               3:  //M003_GENERATE_ALERT
                   #methodInputs := REF("MII_Interface_Data".MII_METHODS."M003_GENERATE_ALERT".Inputs);
                   VariantPut(SRC := "MII_Interface_Data".MII_METHODS."M003_GENERATE_ALERT".Inputs,
                              DST := #methodInputs);
                   #methodOutputs := REF("MII_Interface_Data".MII_METHODS."M003_GENERATE_ALERT".Outputs);
                   VariantPut(SRC := "MII_Interface_Data".MII_METHODS."M003_GENERATE_ALERT".Outputs,
                              DST := #methodOutputs);

               4:  //M102_REWORK_DECLARATION
                   #methodInputs := REF("MII_Interface_Data".MII_METHODS."M102_REWORK_DECLARATION".Inputs);
                   VariantPut(SRC := "MII_Interface_Data".MII_METHODS."M102_REWORK_DECLARATION".Inputs,
                              DST := #methodInputs);
                   #methodOutputs := REF("MII_Interface_Data".MII_METHODS."M102_REWORK_DECLARATION".Outputs);
                   VariantPut(SRC := "MII_Interface_Data".MII_METHODS."M102_REWORK_DECLARATION".Outputs,
                              DST := #methodOutputs);

               5:  //M002_GET_PLANTS
                   #methodOutputs := REF("MII_Interface_Data".MII_METHODS."M002_GET_PLANTS".Outputs);
                   VariantPut(SRC := "MII_Interface_Data".MII_METHODS.M002_GET_PLANTS.Outputs,
                              DST := #methodOutputs);

               6: //NON TRS
                   #methodInputs := REF("MII_Interface_Data".MII_METHODS.M004_NTRS.Inputs);
                   VariantPut(SRC := "MII_Interface_Data".MII_METHODS.M004_NTRS.Inputs,
                              DST := #methodInputs);
                   #methodOutputs := REF("MII_Interface_Data".MII_METHODS.M004_NTRS.Outputs);
                   VariantPut(SRC := "MII_Interface_Data".MII_METHODS.M004_NTRS.Outputs,
                              DST := #methodOutputs);

               7: //PY
                   #methodInputs := REF("MII_Interface_Data".MII_METHODS.M103_PY.Inputs);
                   VariantPut(SRC := "MII_Interface_Data".MII_METHODS.M103_PY.Inputs,
                              DST := #methodInputs);
                   #methodOutputs := REF("MII_Interface_Data".MII_METHODS.M103_PY.Outputs);
                   VariantPut(SRC := "MII_Interface_Data".MII_METHODS.M103_PY.Outputs,
                              DST := #methodOutputs);

               8: //VARABILITY
                   #methodInputs := REF("MII_Interface_Data".MII_METHODS.M005_VARIABILITY.Inputs);
                   VariantPut(SRC := "MII_Interface_Data".MII_METHODS.M005_VARIABILITY.Inputs,
                              DST := #methodInputs);
                   #methodOutputs := REF("MII_Interface_Data".MII_METHODS.M005_VARIABILITY.Outputs);
                   VariantPut(SRC := "MII_Interface_Data".MII_METHODS.M005_VARIABILITY.Outputs,
                              DST := #methodOutputs);


           END_CASE;
       END_REGION ;
   END_IF;
END_REGION

REGION Network 3: Call client fb
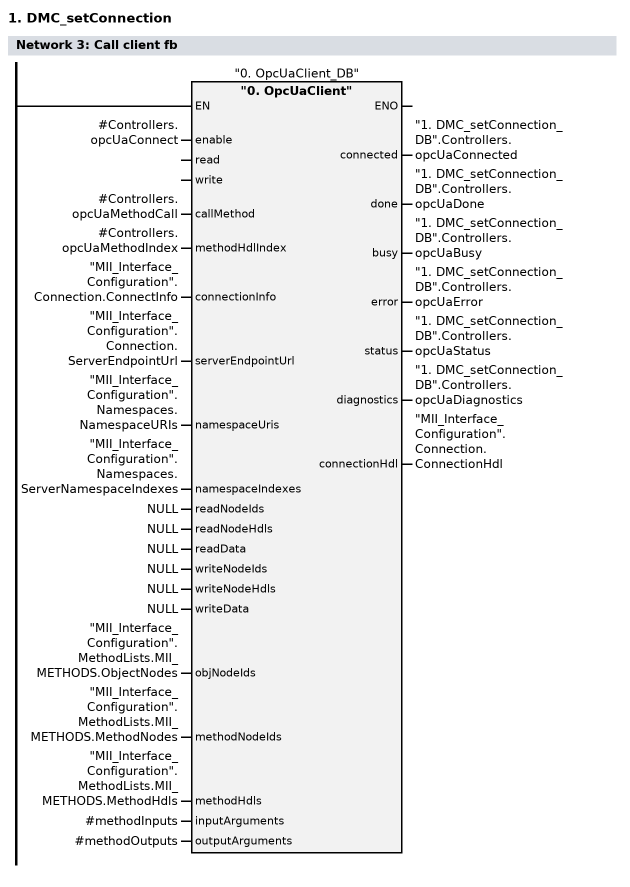
   RUNG wire#powerrail
      "0. OpcUaClient_DB"(enable := #Controllers.opcUaConnect, read :=, write :=, callMethod := #Controllers.opcUaMethodCall, methodHdlIndex := #Controllers.opcUaMethodIndex, connectionInfo := "MII_Interface_Configuration".Connection.ConnectInfo, serverEndpointUrl := "MII_Interface_Configuration".Connection.ServerEndpointUrl, namespaceUris := "MII_Interface_Configuration".Namespaces.NamespaceURIs, namespaceIndexes := "MII_Interface_Configuration".Namespaces.ServerNamespaceIndexes, readNodeIds := NULL, readNodeHdls := NULL, readData := NULL, writeNodeIds := NULL, writeNodeHdls := NULL, writeData := NULL, objNodeIds := "MII_Interface_Configuration".MethodLists.MII_METHODS.ObjectNodes, methodNodeIds := "MII_Interface_Configuration".MethodLists.MII_METHODS.MethodNodes, methodHdls := "MII_Interface_Configuration".MethodLists.MII_METHODS.MethodHdls, inputArguments := #methodInputs, outputArguments := #methodOutputs, connected => "1. DMC_setConnection_DB".Controllers.opcUaConnected, done => "1. DMC_setConnection_DB".Controllers.opcUaDone, busy => "1. DMC_setConnection_DB".Controllers.opcUaBusy, error => "1. DMC_setConnection_DB".Controllers.opcUaError, status => "1. DMC_setConnection_DB".Controllers.opcUaStatus, diagnostics => "1. DMC_setConnection_DB".Controllers.opcUaDiagnostics, connectionHdl => "MII_Interface_Configuration".Connection.ConnectionHdl)
   END_RUNG
   // the same network as SCL:
   "0. OpcUaClient_DB"(enable := #Controllers.opcUaConnect,   // "0. OpcUaClient"
                       callMethod := #Controllers.opcUaMethodCall,
                       methodHdlIndex := #Controllers.opcUaMethodIndex,
                       connectionInfo := "MII_Interface_Configuration".Connection.ConnectInfo,
                       serverEndpointUrl := "MII_Interface_Configuration".Connection.ServerEndpointUrl,
                       namespaceUris := "MII_Interface_Configuration".Namespaces.NamespaceURIs,
                       namespaceIndexes := "MII_Interface_Configuration".Namespaces.ServerNamespaceIndexes,
                       readNodeIds := NULL,
                       readNodeHdls := NULL,
                       readData := NULL,
                       writeNodeIds := NULL,
                       writeNodeHdls := NULL,
                       writeData := NULL,
                       objNodeIds := "MII_Interface_Configuration".MethodLists.MII_METHODS.ObjectNodes,
                       methodNodeIds := "MII_Interface_Configuration".MethodLists.MII_METHODS.MethodNodes,
                       methodHdls := "MII_Interface_Configuration".MethodLists.MII_METHODS.MethodHdls,
                       inputArguments := #methodInputs,
                       outputArguments := #methodOutputs,
                       connected => "1. DMC_setConnection_DB".Controllers.opcUaConnected,
                       done => "1. DMC_setConnection_DB".Controllers.opcUaDone,
                       busy => "1. DMC_setConnection_DB".Controllers.opcUaBusy,
                       error => "1. DMC_setConnection_DB".Controllers.opcUaError,
                       status => "1. DMC_setConnection_DB".Controllers.opcUaStatus,
                       diagnostics => "1. DMC_setConnection_DB".Controllers.opcUaDiagnostics,
                       connectionHdl => "MII_Interface_Configuration".Connection.ConnectionHdl);
END_REGION

REGION Network 4 (SCL): Post method call
   IF #Controllers.opcUaMethodCall AND (#Controllers.opcUaDone OR #Auxiliar.timeout) THEN
       REGION SWITCH CASE
           CASE #Controllers.opcUaMethodIndex OF
               0:  //M000_PRODUCTION_DECLARATION
                   //Send the inputs and the output to the HMI
                   "MII_Parameters".M000_Status.Inputs := "MII_Interface_Data".MII_METHODS.M000_PRODUCTION_DECLARATION.Inputs;
                   "MII_Parameters".M000_Status.Outputs := "MII_Interface_Data".MII_METHODS.M000_PRODUCTION_DECLARATION.Outputs;


                   IF "MII_Interface_Data".MII_METHODS.M000_PRODUCTION_DECLARATION.Outputs.SUCCESS_FLAG = 0 OR #Auxiliar.timeout THEN
                       //Write error status
                       IF #Auxiliar.timeout THEN
                           "MII_Parameters".M000_Status.status := Wstring#'TimeoutERROR';
                       ELSE
                           "MII_Parameters".M000_Status.status := "MII_Interface_Data".MII_METHODS.M000_PRODUCTION_DECLARATION.Outputs.STATUS_MESSAGE;
                       END_IF;

                       //Get error timestamp 
                       #retVal := RD_LOC_T("MII_Parameters".M000_Status.timestamp);

                       //Set error trigger to HMI store values
                       //Note: HMI must reset this tag after writing the file
                       "MII_Parameters".M000_Status.error := TRUE;
                   ELSE
                       //Reset error if declaration is ok
                       "MII_Parameters".M000_Status.error := FALSE;
                       "MII_Parameters".M000_Status.status := "MII_Interface_Data".MII_METHODS.M000_PRODUCTION_DECLARATION.Outputs.STATUS_MESSAGE;
                   END_IF;

                   //Reset test command and add one to the auxiliar cycle counter
                   IF "MII_Parameters".Commands.testProdDeclaration THEN
                       "MII_Parameters".Commands.testProdDeclaration := FALSE;
                       "MII_Parameters".Commands.auxTestProdDeclaration := "MII_Parameters".Commands.auxTestProdDeclaration + 1;
                   END_IF;

               1: //M002_GET_LOCAL_TIME
                   IF #Auxiliar.timeout THEN
                       "MII_Parameters".M002_Status.status := WSTRING#'TimeoutERROR';
                   ELSE
                       //Overwrite system time
                       #retVal := WR_LOC_T(LOCTIME := "MII_Interface_Data".MII_METHODS.M001_GET_LOCAL_TIME.Outputs.DATETIME_LOCAL, DST := TRUE);

                       //Set M002_status
                       "MII_Parameters".M002_Status.localTime := "MII_Interface_Data".MII_METHODS.M001_GET_LOCAL_TIME.Outputs.DATETIME_LOCAL;
                       "MII_Parameters".M002_Status.status := WSTRING#'OK';

                       //Reset command after calling the method
                       "MII_Parameters".Commands.getLocalTime := FALSE;
                   END_IF;

               2: //TO BE DEVELOPED
                   ;

               3: //TO BE DEVELOPED
                   ;

               4: //TO BE DEVELOPED
                   ;

               5: //TO BE DEVELOPED
                   ;

               6: //TO BE DEVELOPED
                   ;

               7: //TO BE DEVELOPED
                   ;

               8: //TO BE DEVELOPED
                   ;

           END_CASE;
       END_REGION

       //RESET METHOD INDEX
       #CallBuffer[#Controllers.opcUaMethodIndex] := FALSE;

       //RESET METHOD TAG
       #Controllers.opcUaMethodCall := FALSE;
   END_IF;
END_REGION

REGION Network 5 (SCL): Device diagnostics
   // Read diagnostic status
   "MII_Parameters".Connection_Status.opcUaConnected := #Controllers.opcUaConnected;
   "MII_Parameters".Connection_Status.opcUaError := #Controllers.opcUaError;
   "MII_Parameters".Connection_Status.opcUaStatus := #Controllers.opcUaStatus;
   "MII_Parameters".Connection_Status.opcUaDiagnostics := #Controllers.opcUaDiagnostics.subfunctionStatus;

   // Shift data to display on HMI
   IF #Controllers.opcUaDiagnostics.subfunctionStatus > 65536 THEN
       "MII_Parameters".Connection_Status.aux.opcUaSubfunctionStatus := SHR(IN := #Controllers.opcUaDiagnostics.subfunctionStatus, N := 16);
   END_IF;

   // Output error parameters
   IF NOT #Controllers.opcUaError THEN
       CASE #Controllers.opcUaStatus OF
           16#0000:
               IF NOT #Controllers.opcUaDone THEN
                   //Client not connected.
                   "MII_Parameters".Connection_Status.aux.diagnosticStatus := 1;
               ELSE
                   //Job successfully executed.
                   "MII_Parameters".Connection_Status.aux.diagnosticStatus := 2;
               END_IF;

           16#7000:
               IF NOT #Controllers.opcUaDone THEN
                   //Client connected and ready for job.
                   "MII_Parameters".Connection_Status.aux.diagnosticStatus := 3;
               ELSE
                   //Connection successfully established and ready for job.
                   "MII_Parameters".Connection_Status.aux.diagnosticStatus := 4;
               END_IF;

           16#7001: //Job is running.
               "MII_Parameters".Connection_Status.aux.diagnosticStatus := 5;
       END_CASE;
   ELSE
       // Output parameters with error
       "MII_Parameters".Connection_Status.aux.diagnosticStatus := #Controllers.opcUaStatus;

       // Automatically manage the 16#80AE_0000 error
       IF NOT "MII_Parameters".Commands.forceReconnection AND NOT "MII_Parameters".Connection_Status.opcUaConnected THEN
           // Forces the reconnection
           "MII_Parameters".Commands.forceReconnection := TRUE;

           IF "0. OpcUaClient_DB".statOpcUaRequests.disconnect THEN
               // Reset disconnect button 
               "0. OpcUaClient_DB".statOpcUaRequests.disconnect := FALSE;
           END_IF;
       END_IF;
   END_IF;
END_REGION

REGION Network 6 (SCL): Try to call method again routine
   // //Method call timeout
   // #Timers.tryAgain(IN := "MII_Parameters".M000_Status.error,
   //                  PT := t#2s,
   //                  Q => #Auxiliar.tryAgain);

   // IF #Controllers.opcUaConnected AND #Auxiliar.tryAgain THEN
   //              //Try again
   //              IF NOT #CallBuffer[0] THEN
   //                  #CallBuffer[0] := TRUE;

   //                  //Add one attempt to counter
   //                  "MII_Parameters".Connection_Status.aux.nAttemptsTotal := "MII_Parameters".Connection_Status.aux.nAttemptsTotal + 1;
   //              END_IF;

   //              //Restart timer
   //              RESET_TIMER(#Timers.tryAgain);

   //          END_IF;
END_REGION
END_FUNCTION_BLOCK

FUNCTION_BLOCK "0. OpcUaClient"
TITLE = OpcUaClient
{ S7_Optimized_Access := 'FALSE' }
AUTHOR : SiemensAG
VERSION : 1.3
//OPC UA-Client-Wrapper
   VAR_INPUT 
      enable : Bool;   // TRUE: Enable connection to OPC UA server
      read : Bool;   // TRUE: Execute Read functionality
      write : Bool;   // TRUE: Execute Write functionality
      callMethod : Bool;   // TRUE: Execute Method Call
      methodHdlIndex : SInt;   // Index of method in "methodHdls" that should be called
      connectionInfo {InstructionName := 'OPC_UA_SessionConnectInfo'; LibVersion := '1.0'} : OPC_UA_SessionConnectInfo;   // Connection Information for session establishment to OPC UA server
      serverEndpointUrl : String;   // Endpoint of OPC UA server
   END_VAR

   VAR_OUTPUT 
      connected { ExternalWritable := 'False'} : Bool;   // TRUE: Connection to OPC UA server is established and valid
      done { ExternalWritable := 'False'} : Bool;   // TRUE: Functions Read, Write or Method Call were executed successfully
      busy { ExternalWritable := 'False'} : Bool;   // TRUE: FB is working
      error { ExternalWritable := 'False'} : Bool;   // TRUE: FB is in faulty state
      status { ExternalWritable := 'False'} : Word;   // 16#0000 - 16#7FFF: Status of the FB, 16#8000 - 16#FFFF: Error identification
      diagnostics { ExternalWritable := 'False'} : "typeFbDiagnostics";   // Diagnostics information of FB when error occurs
      connectionHdl { ExternalWritable := 'False'} : DWord;   // Connection handle which is used for OPC UA connection to the server
   END_VAR

   VAR_IN_OUT 
      namespaceUris : Variant;   // Pointer to the Namespace URIs of the OPC UA client interface (NULL if not used)
      namespaceIndexes : Variant;   // Pointer to the Namespace Indexes of the OPC UA client interface (NULL if not used)
      readNodeIds : Variant;   // Pointer to the Node-IDs of the nodes to read of the OPC UA client interface (NULL if not used)
      readNodeHdls : Variant;   // Pointer to the Node handles of the registered nodes to read of the OPC UA client interface (NULL if not used)
      readData : Variant;   // Pointer to the storage area for read data (NULL if not used)
      writeNodeIds : Variant;   // Pointer to the Node-IDs of the nodes to write of the OPC UA client interface (NULL if not used)
      writeNodeHdls : Variant;   // Pointer to the Node handles of the registered nodes to write of the OPC UA client interface (NULL if not used)
      writeData : Variant;   // Pointer to the storage area for write data (NULL if not used)
      objNodeIds : Variant;   // Pointer to the Node-IDs of the method objects (instance DB) of the OPC UA client interface (NULL if not used)
      methodNodeIds : Variant;   // Pointer to the Node-IDs of the methods of the OPC UA client Interface (NULL if not used)
      methodHdls : Variant;   // Pointer to the Node handles of the registered methods of the OPC UA client interface (NULL if not used)
      inputArguments : Variant;   // Pointer to the Input Arguments of the called method (NULL if not used)
      outputArguments : Variant;   // Pointer to the Output Arguments of the called method (NULL if not used)
   END_VAR

   VAR 
      instOpcUaConnect {InstructionName := 'OPC_UA_Connect'; LibVersion := '1.0'; ExternalAccessible := 'False'; ExternalVisible := 'False'; ExternalWritable := 'False'} : OPC_UA_Connect;
      instOpcUaConnectionGetStatus {InstructionName := 'OPC_UA_ConnectionGetStatus'; LibVersion := '1.0'; ExternalAccessible := 'False'; ExternalVisible := 'False'; ExternalWritable := 'False'} : OPC_UA_ConnectionGetStatus;
      instOpcUaNamespaceGIL {InstructionName := 'OPC_UA_NamespaceGetIndexList'; LibVersion := '1.0'; ExternalAccessible := 'False'; ExternalVisible := 'False'; ExternalWritable := 'False'} : OPC_UA_NamespaceGetIndexList;
      InstOpcUaGHLRead {InstructionName := 'OPC_UA_NodeGetHandleList'; LibVersion := '1.0'; ExternalAccessible := 'False'; ExternalVisible := 'False'; ExternalWritable := 'False'} : OPC_UA_NodeGetHandleList;
      instOpcUaGHLWrite {InstructionName := 'OPC_UA_NodeGetHandleList'; LibVersion := '1.0'; ExternalAccessible := 'False'; ExternalVisible := 'False'; ExternalWritable := 'False'} : OPC_UA_NodeGetHandleList;
      instOpcUaGHLMethods {InstructionName := 'OPC_UA_MethodGetHandleList'; LibVersion := '1.0'; ExternalAccessible := 'False'; ExternalVisible := 'False'; ExternalWritable := 'False'} : OPC_UA_MethodGetHandleList;   // Get node handles for Methods
      InstOpcUaRHLRead {InstructionName := 'OPC_UA_NodeReleaseHandleList'; LibVersion := '1.0'; ExternalAccessible := 'False'; ExternalVisible := 'False'; ExternalWritable := 'False'} : OPC_UA_NodeReleaseHandleList;
      instOpcUaRHLWrite {InstructionName := 'OPC_UA_NodeReleaseHandleList'; LibVersion := '1.0'; ExternalAccessible := 'False'; ExternalVisible := 'False'; ExternalWritable := 'False'} : OPC_UA_NodeReleaseHandleList;
      instOpcUaRHLMethods {InstructionName := 'OPC_UA_MethodReleaseHandleList'; LibVersion := '1.0'; ExternalAccessible := 'False'; ExternalVisible := 'False'; ExternalWritable := 'False'} : OPC_UA_MethodReleaseHandleList;
      instOpcUaReadList {InstructionName := 'OPC_UA_ReadList'; LibVersion := '1.0'; ExternalAccessible := 'False'; ExternalVisible := 'False'; ExternalWritable := 'False'} : OPC_UA_ReadList;
      instOpcUaWriteList {InstructionName := 'OPC_UA_WriteList'; LibVersion := '1.0'; ExternalAccessible := 'False'; ExternalVisible := 'False'; ExternalWritable := 'False'} : OPC_UA_WriteList;   // Write values of multiple nodes
      instOpcUaMethodCall {InstructionName := 'OPC_UA_MethodCall'; LibVersion := '1.0'; ExternalAccessible := 'False'; ExternalVisible := 'False'; ExternalWritable := 'False'} : OPC_UA_MethodCall;
      instOpcUaDisconnect {InstructionName := 'OPC_UA_Disconnect'; LibVersion := '1.0'; ExternalAccessible := 'False'; ExternalVisible := 'False'; ExternalWritable := 'False'} : OPC_UA_Disconnect;
      statOldTriggers { ExternalAccessible := 'False'; ExternalVisible := 'False'; ExternalWritable := 'False'} : Struct   // Internal structure for Trigger handling
         connect { ExternalAccessible := 'False'; ExternalVisible := 'False'; ExternalWritable := 'False'} : Bool;   // Saved Trigger for Connection establishment
         reconnect { ExternalAccessible := 'False'; ExternalVisible := 'False'; ExternalWritable := 'False'} : Bool;   // Saved Trigger for Connection reestablishment
         disconnect { ExternalAccessible := 'False'; ExternalVisible := 'False'; ExternalWritable := 'False'; S7_SetPoint := 'True'} : Bool;   // Saved Trigger for disconnecting
         read { ExternalAccessible := 'False'; ExternalVisible := 'False'; ExternalWritable := 'False'; S7_SetPoint := 'True'} : Bool;   // Saved Trigger for Read
         write { ExternalAccessible := 'False'; ExternalVisible := 'False'; ExternalWritable := 'False'; S7_SetPoint := 'True'} : Bool;   // Saved Trigger for Write
         callMethod { ExternalAccessible := 'False'; ExternalVisible := 'False'; ExternalWritable := 'False'} : Bool;   // Saved Trigger for Method Call
         clearSession { ExternalAccessible := 'False'; ExternalVisible := 'False'; ExternalWritable := 'False'} : Bool;   // Saved Trigger for Session Clearing
      END_STRUCT;
      statState { ExternalWritable := 'False'} : Int;   // Actual state of the state machine. 0: connect; 1: get Namespaces; 3: Get List Handles; 4: Connected; 5: Disconnect
      statDone { ExternalAccessible := 'False'; ExternalVisible := 'False'; ExternalWritable := 'False'} : Bool;   // Read, Write, MethodCall finished without error.
      statConnected { ExternalAccessible := 'False'; ExternalVisible := 'False'; ExternalWritable := 'False'} : Bool;   // Connection to OPC UA Server is established and valid.
      statBusy { ExternalVisible := 'False'; ExternalWritable := 'False'} : Bool;   // FB is busy.
      statDiagnostics { ExternalAccessible := 'False'; ExternalVisible := 'False'; ExternalWritable := 'False'} : "typeFbDiagnostics";   // Diagnostic structure for internal use.
      statDiagnosticsEmpty { ExternalWritable := 'False'} : "typeFbDiagnostics";   // Empty diagnostic structure, to initialize Output.
      statOpcUaRequests { ExternalAccessible := 'False'; ExternalVisible := 'False'; ExternalWritable := 'False'} : Struct   // Internal structure for OPC UA function blocks requests.
         connect { ExternalAccessible := 'False'; ExternalVisible := 'False'; ExternalWritable := 'False'} : Bool;   // Request for OPC_UA_Connect
         conGS { ExternalAccessible := 'False'; ExternalVisible := 'False'; ExternalWritable := 'False'} : Bool;   // Request for OPC_UA_ConnectionGetStatus
         NGIL { ExternalAccessible := 'False'; ExternalVisible := 'False'; ExternalWritable := 'False'} : Bool;   // Request for OPC_UA_NamespaceGetIndexList
         readGHL { ExternalAccessible := 'False'; ExternalVisible := 'False'; ExternalWritable := 'False'} : Bool;   // Request for OPC_UA_NodeGetHandleList for ReadList
         methodsGHL { ExternalAccessible := 'False'; ExternalVisible := 'False'; ExternalWritable := 'False'} : Bool;   // Request for OPC_UA_MethodGetHandleList
         writeGHL { ExternalAccessible := 'False'; ExternalVisible := 'False'; ExternalWritable := 'False'} : Bool;   // Request for OPC_UA_NodeGetHandleList for WriteList
         read { ExternalAccessible := 'False'; ExternalVisible := 'False'; ExternalWritable := 'False'} : Bool;   // Request for OPC_UA_ReadList
         write { ExternalAccessible := 'False'; ExternalVisible := 'False'; ExternalWritable := 'False'} : Bool;   // Request for OPC_UA_WriteList
         methodCall { ExternalAccessible := 'False'; ExternalVisible := 'False'; ExternalWritable := 'False'} : Bool;   // Request for OPC_UA_MethodCall
         readRHL { ExternalAccessible := 'False'; ExternalVisible := 'False'; ExternalWritable := 'False'} : Bool;   // Request for OPC_UA_NodeReleaseHandleList for ReadList
         writeRHL { ExternalAccessible := 'False'; ExternalVisible := 'False'; ExternalWritable := 'False'} : Bool;   // Request for OPC_UA_NodeReleaseHandleList for WriteList
         methodsRHL { ExternalAccessible := 'False'; ExternalVisible := 'False'; ExternalWritable := 'False'} : Bool;   // Request for OPC_UA_MethodReleaseHandleList
         disconnect { ExternalAccessible := 'False'; ExternalVisible := 'False'; ExternalWritable := 'False'} : Bool;   // Request for OPC_UA_Disconnect
      END_STRUCT;
      statRegisteredLists { ExternalWritable := 'False'} : Struct   // Internal structure for registered Lists/Namespaces. For Diagnostic purpose.
         NamespaceIndexes { ExternalWritable := 'False'} : Bool;   // Namespace Indexes are registered by OPC_UA_NamespaceGetIndexList
         Read { ExternalWritable := 'False'} : Bool;   // Read list is registered by OPC_UA_NodeGetHandleList
         Write { ExternalWritable := 'False'} : Bool;   // Write list is registered by OPC_UA_NodeGetHandleList
         Methods { ExternalWritable := 'False'} : Bool;   // Method list is registered by OPC_UA_MethodGetHandleList
      END_STRUCT;
      statDiagCounter { ExternalWritable := 'False'} : Struct   // Internal structure for counting connects/registrations/functions. For Diagnostic purpose.
         Connect { ExternalVisible := 'False'; ExternalWritable := 'False'} : UInt;   // Counter for successful connects or reconnects.
         NamespaceReg { ExternalWritable := 'False'} : UInt;   // Counter for successful Namespace registrations.
         RegisterRead { ExternalWritable := 'False'} : UInt;   // Counter for successful Read List registrations.
         RegisterWrite { ExternalWritable := 'False'} : UInt;   // Counter for successful Write List registrations.
         RegisterMethods { ExternalWritable := 'False'} : UInt;   // Counter for successful Method List registrations.
         Read { ExternalWritable := 'False'} : UInt;   // Counter for successful Read function executions.
         Write { ExternalWritable := 'False'} : UInt;   // Counter for successful Write function executions.
         MethodCall { ExternalWritable := 'False'} : UInt;   // Counter for successful Method Calls.
      END_STRUCT;
      statMethodResult { ExternalWritable := 'False'} : DWord;   // OPC UA result after Method Call.
      statMethodHdl { ExternalAccessible := 'False'; ExternalVisible := 'False'; ExternalWritable := 'False'} : DWord;   // Calculated Method Handle. Dependend on INPUT: methodHdlIndex.
      statMethodHdlId { ExternalAccessible := 'False'; ExternalVisible := 'False'; ExternalWritable := 'False'} : DInt;   // Internal Variable for INPUT: methodHdlIndex.
      statConnectionHdl { ExternalAccessible := 'False'; ExternalVisible := 'False'; ExternalWritable := 'False'} : DWord;   // Internal Variable for Connection Handle.
      statRHLTrigger { ExternalAccessible := 'False'; ExternalVisible := 'False'; ExternalWritable := 'False'} : Bool;   // Trigger, do start with releasing Lists for disconnect.
      statCheckConnectionStatus { ExternalAccessible := 'False'; ExternalVisible := 'False'; ExternalWritable := 'False'} : Bool;   // If TRUE, OPC_UA_ConnectionGetStatus is called to diagnose the connection.
      statCycDiagTrigger { ExternalAccessible := 'False'; ExternalVisible := 'False'; ExternalWritable := 'False'} : Bool;   // Cyclic trigger for OPC_UA_ConnectionGetStatus-
      instCycDiag {InstructionName := 'IEC_TIMER'; LibVersion := '1.0'; ExternalAccessible := 'False'; ExternalVisible := 'False'; ExternalWritable := 'False'} : IEC_TIMER;   // Timer for cyclic connection diagnostics.
      statOpcUaReadTimeStamps { ExternalWritable := 'False'} : Array[0..299] of LDT;   // Timestamps of read variables. For diagnostic purpose.
      statSerializeMethodHdls { ExternalAccessible := 'False'; ExternalVisible := 'False'; ExternalWritable := 'False'} : Array[0..1199] of Byte;   // Array for calculating the MethodHdl together with the INPUT methodHdlIndex.
      statOpcUaStatusLists { ExternalWritable := 'False'} : Struct   // Internal structure for Status Lists, that are used by every OPC_UA_xxx FB
         methodRHL { ExternalWritable := 'False'} : Array[0..299] of DWord;   // Status List for Method OPC_UA_ReleaseHandleList
         methodGHL { ExternalWritable := 'False'} : Array[0..299] of DWord;   // Status List for Method OPC_UA_GetHandleList
         writeRHL { ExternalWritable := 'False'} : Array[0..299] of DWord;   // Status List for Write OPC_UA_ReleaseHandleList
         writeList { ExternalWritable := 'False'} : Array[0..299] of DWord;   // Status List for Write OPC_UA_WritedList
         writeGHL { ExternalWritable := 'False'} : Array[0..299] of DWord;   // Status List for WriteOPC_UA_GetHandleList
         readRHL { ExternalWritable := 'False'} : Array[0..299] of DWord;   // Status List for Read OPC_UA_ReleaseHandleList
         readList { ExternalWritable := 'False'} : Array[0..299] of DWord;   // Status List for Read OPC_UA_ReadList
         readGHL { ExternalWritable := 'False'} : Array[0..299] of DWord;   // Status List for Read OPC_UA_GetHandleList
         namespaceGIL { ExternalWritable := 'False'} : Array[0..299] of DWord;   // Status List for Namespace OPC_UA_NamespaceGetIndexList
      END_STRUCT;
   END_VAR

   VAR_TEMP 
      tempIndex : Int;   // Index for finding errors in statOpcUaStatusLists.
      tempRetVal : Int;   // Return value for Serialize function, that is used for calculating statMethodHdl.
      tempConnectTrigger : Bool;   // Temporary trigger for connection establishment.
      tempDisconnectTrigger : Bool;   // Temporary trigger for disconnect.
      tempReadTrigger : Bool;   // Temporary trigger for Read function.
      tempWriteTrigger : Bool;   // Temporary trigger for Write function.
      tempMethodCallTrigger : Bool;   // Temporary trigger for Method Calls.
      tempReconnectTrigger : Bool;   // Temporary trigger for reconnect.
      tempClearSessionTrigger : Bool;   // Temporary trigger for clean up Session.
   END_VAR

   VAR CONSTANT 
      STATE_CONNECT : Int := 0;   // State for idling until INPUT enable is triggered, to establish a connection.
      STATE_NAMESPACE_GET_INDEX_LIST : Int := 1;   // State for getting Namespace indexes.
      STATE_NODE_GET_HANDLE_LIST : Int := 3;   // State for registration of Read/Write/Method Lists
      STATE_CONNECTED : Int := 4;   // State for idling until INPUT read/write/methodCall has positive edge, to execute function.
      STATE_DISCONNECT : Int := 5;   // State for releasing Read/Write/Method Lists and disconnect.
      CGS_CONNECTED : UDInt := 0;   // OPC_UA_ConnectionGetStatus Connection state is connected.
      CGS_CONN_ERROR : UDInt := 1;   // OPC_UA_ConnectionGetStatus Connection state is in error.
      CGS_SHUTDOWN : UDInt := 2;   // OPC_UA_ConnectionGetStatus Connection state is in shutdown, nodes have to be released and connection terminated.
      CGS_SS_RUNNING : UDInt := 0;   // OPC_UA_ConnectionGetStatus Server state is running.
      CGS_SL_GOOD : Byte := 16#FF;   // OPC_UA_ConnectionGetStatus Connection state is connected.
      STATUS_SESSION_CLEANEDUP : DWord := 16#A000_0105;   // OPC_UA_ConnectionGetStatus: Session is cleaned up and has to be reconnected.
      STATUS_SERVER_NOT_CONNECTED : DWord := 16#800D_0000;   // OPC_UA_ConnectionGetStatus: Choosen Server is not connected.
      STATUS_BAD_CONNECTION_CLOSED : DWord := 16#80AE_0000;   // OPC_UA_ConnectionGetStatus
      STATUS_BUSY : Word := 16#7001;   // Function block is busy.
      STATUS_IDLE : Word := 16#7000;   // Function block idles.
      STATUS_NOT_REGISTERED : Word := 16#80FF;   // Read/Write/Method List is not registered
      STATUS_DONE : Word := 16#0000;   // Read/Write/Method Call was successfully executed.
      CYC_TIME_GCS : Time := T#5S;   // Time for cylic call of OPC_UA_ConnectionGetStatus
      OPC_UA_FUNCTIONS_TIMEOUT : Time := T#10S;   // Timout for all OPC UA Client Function blocks
      ERR_CONNECT : Word := 16#8601;   // Error during connect.
      ERR_NGIL : Word := 16#8602;   // Error during getting Namespace Indexes
      ERR_NGIL_SL : Word := 16#8617;   // Error in Namespace indexes Status list
      ERR_R_GHL : Word := 16#8631;   // Error during Read list registration
      ERR_R_GHL_SL : Word := 16#8731;   // Error in Read handle list Status list
      ERR_W_GHL : Word := 16#8632;   // Error during Write list registration
      ERR_W_GHL_SL : Word := 16#8732;   // Error in Write handle list Status list
      ERR_M_GHL : Word := 16#8633;   // Error during Method list registration
      ERR_M_GHL_SL : Word := 16#8733;   // Error in Method handle List status list
      ERR_RL : Word := 16#8604;   // Error during Read List execution
      ERR_RL_NOTREG : Word := 16#86F4;   // Error, because no Read List is registered, but Read execution was triggered
      ERR_RL_SL : Word := 16#8614;   // Error in Read list status list.
      ERR_WL : Word := 16#8605;   // Error during Write List execution
      ERR_WL_NOTREG : Word := 16#86F5;   // Error, because no Write List is registered, but Write execution was triggered
      ERR_WL_SL : Word := 16#8615;   // Error in Write list status list
      ERR_MC : Word := 16#8606;   // Error durging Method Call execution
      ERR_MC_NOTREG : Word := 16#86F6;   // Error, because no Method List is registered, but Method call execution was triggered
      ERR_MC_SERIALIZE : Word := 16#8616;   // Error during MethodHdl calculation, in Serialize function
      ERR_MC_RESULT : Word := 16#8626;   // Error, that was reported by Methods OPC UA result
      ERR_R_RHL : Word := 16#8671;   // Error during release of Read List
      ERR_R_RHL_SL : Word := 16#8771;   // Error in Release Read List status list
      ERR_W_RHL : Word := 16#8672;   // Error during realease of Write list
      ERR_W_RHL_SL : Word := 16#8772;   // Error in Release Write List status list
      ERR_M_RHL : Word := 16#8673;   // Error during relaese of Method List
      ERR_M_RHL_SL : Word := 16#8773;   // Error in Release Method List status List
      ERR_DISCON : Word := 16#8608;   // Error during disconnect.
      ERR_CGS : Word := 16#8610;   // Error in OPC_UA_ConnectionGetStatus
      ERR_CGS_CSTATE : Word := 16#8611;   // Error in OPC_UA_ConnectionGetStatus, regarding Connection Status
      ERR_CGS_CSTATE_SHUTDOWN : Word := 16#8711;   // Error in OPC_UA_ConnectionGetStats, Connection was shut down
      ERR_CGS_SSTATE : Word := 16#8612;   // Error in OPC_UA_ConnectionGetStatus, regarding Server State
      ERR_CGS_SLVL : Word := 16#8613;   // Error in OPC_UA_ConnectionGetStatus, regarding Service Level
      MAX_LIST_LENGTH : UInt := 299;   // Maximum lenth of Write/Readlist
      MAX_LENGTH_METHOD_INDEX : UInt := 399;   // maximum length of MethodHdls (mas 100 Methods per MethodList)
   END_VAR


BEGIN
	//=============================================================================
	// Siemens AG (c)Copyright (2019)
	//-----------------------------------------------------------------------------
	// Library: -
	// Tested with: CPU 1516-3 PN/DP;  FW 2.8
	// Engineering: TIA Portal (V16)
	// Restrictions: -
	// Requirements: OPC UA Client activated, Fimware V2.8; Set PLC time
	// Functionality: Encapsulates OPC UA client blocks for read, write and method
	//                call including connection handling and diagnosis
	//-----------------------------------------------------------------------------
	// Change log table:
	// Version    Date         Expert in charge           Changes applied
	// 01.00.00   01.02.2019   Siemens SUP Applications   First released version
	// 01.01.00   31.11.2019   Siemens SUP Applications   Interface, Styleguide and user program performance changes
	// 01.02.00   15.10.2020   Siemens SUP Applications   Bugfixes
	// 01.03.00   28.07.2021   Siemens SUP Applications   Fixed RHL issues
	//=============================================================================
	
	
	//State machine
	CASE #statState OF
	  #STATE_CONNECT:
	    REGION Connection Handling
	      //initialize FB
	      IF NOT #enable THEN
	        #statBusy := FALSE;
	        #statDone := FALSE;
	        #statDiagnostics := #statDiagnosticsEmpty;
	        #statOldTriggers.connect := FALSE;
	        #statConnected := FALSE;
	        #statDiagnostics.status := #STATUS_DONE;
	      END_IF;
	      
	      //Rising Edge detection of connect
	      #tempConnectTrigger := #enable AND NOT #statOldTriggers.connect;
	      #statOldTriggers.connect := #enable;
	      //Rising Edge detection for Reconnect functionality
	      #tempReconnectTrigger := #enable AND NOT #statConnected
	      // AND (#statDiagnostics.subfunctionStatus = #STATUS_SESSION_CLEANEDUP
	      // OR #statDiagnostics.subfunctionStatus = #STATUS_BAD_CONNECTION_CLOSED)
	      AND #statDiagnostics.subfunctionStatus = UDINT_TO_DWORD(#CGS_SHUTDOWN)
	      AND NOT #statOldTriggers.reconnect;
	      #statOldTriggers.reconnect := #enable AND NOT #statConnected
	      // AND (#statDiagnostics.subfunctionStatus = #STATUS_SESSION_CLEANEDUP
	      // OR #statDiagnostics.subfunctionStatus = #STATUS_BAD_CONNECTION_CLOSED);
	      AND #statDiagnostics.subfunctionStatus = UDINT_TO_DWORD(#CGS_SHUTDOWN);
	      
	      //If Connect requested, start connection establishment
	      //---------CONNECT HANDLING-------------
	      //--------------------------------------
	      IF #tempConnectTrigger OR #tempReconnectTrigger THEN
	        IF #statConnectionHdl = 16#0 THEN
	          // no connectionHdl is used -> ready to connect
	          #statOpcUaRequests.connect := TRUE;
	          // set FB outputs
	          #statBusy := TRUE;
	          #statDiagnostics.status := #STATUS_BUSY;
	        ELSE
	          //connectionHdl might be defect, first delete connectionHdl
	          //-> not ready to connect
	          #statOpcUaRequests.disconnect := TRUE;
	          //set FB Outputs
	          #statBusy := TRUE;
	          #statDiagnostics.status := #STATUS_BUSY;
	        END_IF;
	      ELSE
	        IF #instOpcUaDisconnect.Error OR #instOpcUaDisconnect.Done AND #enable THEN
	          //possibly open connection handle is not available or is disconnected
	          //-> ready to connect
	          #statOpcUaRequests.disconnect := FALSE;
	          #statOpcUaRequests.connect := TRUE;
	          #statConnectionHdl := 0;
	        ELSE
	          //nothing done by OPC UA Disconnect block -> Not ready to connect
	          #statOpcUaRequests.connect := FALSE;
	        END_IF;
	      END_IF;
	      
	      //Error at connection establishment
	      IF #instOpcUaConnect.Error THEN
	        #statDone := FALSE;
	        #statConnected := FALSE;
	        #statDiagnostics.status := #ERR_CONNECT;
	        #statDiagnostics.subfunctionStatus := #instOpcUaConnect.Status;
	      END_IF;
	      
	      //Connection establishment was successful
	      IF #instOpcUaConnect.Done THEN
	        #statConnected := TRUE;
	        #statOldTriggers.reconnect := FALSE;
	        #statDiagCounter.Connect += 1;
	        #statState := #STATE_NAMESPACE_GET_INDEX_LIST;
	      END_IF;
	      
	    END_REGION
	    
	  #STATE_NAMESPACE_GET_INDEX_LIST:
	    REGION Handle Namespaces
	      //Request Namespace get Indexlist
	      #statOpcUaRequests.NGIL := TRUE;
	      #statDiagnostics.status := #STATUS_BUSY;
	      
	      // Get Index List was not successful
	      IF #instOpcUaNamespaceGIL.Error THEN
	        //--> Call ConnectionGetStatus if Status = "16#800D0000"
	        IF #instOpcUaNamespaceGIL.Status = #STATUS_SERVER_NOT_CONNECTED THEN
	          #statCheckConnectionStatus := TRUE;
	        ELSE
	          #statState := #STATE_CONNECT;
	        END_IF;
	        #statOpcUaRequests.NGIL := FALSE;
	        // => OUT
	        #statBusy := FALSE;
	        #statDiagnostics.status := #ERR_NGIL;
	        #statDiagnostics.subfunctionStatus := #instOpcUaNamespaceGIL.Status;
	      END_IF;
	      
	      //Get Index List was successful
	      IF #instOpcUaNamespaceGIL.Done THEN
	        //Check StatusList
	        FOR #tempIndex := 0 TO UDINT_TO_INT(CountOfElements(#namespaceUris) - 1) DO
	          IF #statOpcUaStatusLists.#namespaceGIL[#tempIndex] <> 16#0 THEN
	            #statOpcUaRequests.NGIL := FALSE;
	            // => OUT
	            #statDiagnostics.status := #ERR_NGIL_SL;
	            #statDiagnostics.subfunctionStatus := #statOpcUaStatusLists.namespaceGIL[#tempIndex];
	            // error during NGIL call --> connection establishment failed
	            #statState := #STATE_CONNECT;
	            EXIT;
	          END_IF;
	        END_FOR;
	        #statOpcUaRequests.NGIL := FALSE;
	        IF NOT #statDiagnostics.status.%X15 THEN
	          //Count up statNamespaceGetIndexCount
	          #statDiagCounter.NamespaceReg += 1;
	          //statNamespaceIndexesSet
	          #statRegisteredLists.NamespaceIndexes := TRUE;
	          //=>OUT
	          //Next Step
	          #statState := #STATE_NODE_GET_HANDLE_LIST;
	        ELSE
	          #statCheckConnectionStatus := TRUE;
	        END_IF;
	      END_IF;
	    END_REGION
	    
	  #STATE_NODE_GET_HANDLE_LIST:
	    REGION Handle NodeId lists
	      //Trigger NodeHandleList SFBs
	      IF NOT #statRegisteredLists.Write AND #writeNodeIds <> NULL AND #writeNodeHdls <> NULL THEN
	        #statOpcUaRequests.writeGHL := TRUE;
	        #statDiagnostics.status := #STATUS_BUSY;
	      ELSE
	        IF NOT #statRegisteredLists.Read AND #readNodeIds <> NULL AND #readNodeHdls <> NULL THEN
	          #statOpcUaRequests.readGHL := TRUE;
	          #statDiagnostics.status := #STATUS_BUSY;
	        ELSE
	          IF NOT #statRegisteredLists.Methods AND #methodNodeIds <> NULL AND #methodHdls <> NULL AND #objNodeIds <> NULL THEN
	            #statOpcUaRequests.methodsGHL := TRUE;
	            #statDiagnostics.status := #STATUS_BUSY;
	          ELSE
	            #statState := #STATE_CONNECTED;
	            #statBusy := FALSE;
	            #statDiagnostics.status := #STATUS_IDLE;
	          END_IF;
	        END_IF;
	      END_IF;
	      
	      REGION Handle ReadList
	        //Read Node Get Handle List was not successful
	        IF #InstOpcUaGHLRead.Error THEN
	          //--> Call ConnectionGetStatus if Status = "16#800D0000"
	          IF #InstOpcUaGHLRead.Status = #STATUS_SERVER_NOT_CONNECTED THEN
	            #statCheckConnectionStatus := TRUE;
	          ELSE
	            //#statCase := #STATE_CONNECT;
	            #statState := #STATE_CONNECTED;
	          END_IF;
	          #statOpcUaRequests.readGHL := FALSE;
	          // => OUT
	          #statDiagnostics.status := #ERR_R_GHL;
	          #statDiagnostics.subfunctionStatus := #InstOpcUaGHLRead.Status;
	        END_IF;
	        
	        //Read Node Get Handle List was successful
	        IF #InstOpcUaGHLRead.Done THEN
	          //Check StatusList
	          FOR #tempIndex := 0 TO UDINT_TO_INT(CountOfElements(#readNodeIds) - 1) DO
	            IF #statOpcUaStatusLists.#readGHL[#tempIndex] <> 16#0 THEN
	              // => OUT
	              #statBusy := FALSE;
	              #statDiagnostics.status := #ERR_R_GHL_SL;
	              #statDiagnostics.subfunctionStatus := #statOpcUaStatusLists.#readGHL[#tempIndex];
	              EXIT;
	            END_IF;
	          END_FOR;
	          #statOpcUaRequests.readGHL := FALSE;
	          // Count up statRegisterCount
	          #statDiagCounter.RegisterRead += 1;
	          // Nodes are registered
	          #statRegisteredLists.Read := TRUE;
	        END_IF;
	      END_REGION
	      REGION Handle Write List
	        //Write Node Get Handle List was not successful
	        IF #instOpcUaGHLWrite.Error THEN
	          //--> Call ConnectionGetStatus if Status = "16#800D0000"
	          IF #instOpcUaGHLWrite.Status = #STATUS_SERVER_NOT_CONNECTED THEN
	            #statCheckConnectionStatus := TRUE;
	          ELSE
	            //#statCase := #STATE_CONNECT;
	            #statState := #STATE_CONNECTED;
	          END_IF;
	          #statOpcUaRequests.writeGHL := FALSE;
	          // => OUT
	          #statDiagnostics.status := #ERR_W_GHL;
	          #statDiagnostics.subfunctionStatus := #instOpcUaGHLWrite.Status;
	        END_IF;
	        
	        //Write Node Get Handle List was successful
	        IF #instOpcUaGHLWrite.Done THEN
	          //Check StatusList
	          FOR #tempIndex := 0 TO UDINT_TO_INT(CountOfElements(#writeNodeIds) - 1) DO
	            IF #statOpcUaStatusLists.#writeGHL[#tempIndex] <> 16#0 THEN
	              // => OUT
	              #statBusy := FALSE;
	              #statDiagnostics.status := #ERR_W_GHL_SL;
	              #statDiagnostics.subfunctionStatus := #statOpcUaStatusLists.#writeGHL[#tempIndex];
	              //#statCase := #STATE_CONNECT;
	              EXIT;
	            END_IF;
	          END_FOR;
	          #statOpcUaRequests.writeGHL := FALSE;
	          // Count up statRegisterCount
	          #statDiagCounter.RegisterWrite += 1;
	          // Nodes are registered
	          #statRegisteredLists.Write := TRUE;
	        END_IF;
	      END_REGION
	      
	      REGION Handle MethodList
	        //Method Get HandleList was not successful
	        IF #instOpcUaGHLMethods.Error THEN
	          //--> Call ConnectionGetStatus if Status = "16#800D0000"
	          IF #instOpcUaGHLMethods.Status = #STATUS_SERVER_NOT_CONNECTED THEN
	            #statCheckConnectionStatus := TRUE;
	          ELSE
	            //#statCase := #STATE_CONNECT;
	            #statState := #STATE_CONNECTED;
	          END_IF;
	          #statOpcUaRequests.methodsGHL := FALSE;
	          // => OUT
	          #statDiagnostics.status := #ERR_M_GHL;
	          #statDiagnostics.subfunctionStatus := #instOpcUaGHLMethods.Status;
	        END_IF;
	        
	        //Method Get Handle List was successful
	        IF #instOpcUaGHLMethods.Done THEN
	          //Check StatusList
	          FOR #tempIndex := 0 TO UDINT_TO_INT(CountOfElements(#methodNodeIds) - 1) DO
	            IF #statOpcUaStatusLists.#methodGHL[#tempIndex] <> 16#0 THEN
	              // => OUT
	              #statBusy := FALSE;
	              #statDiagnostics.status := #ERR_M_GHL_SL;
	              #statDiagnostics.subfunctionStatus := #statOpcUaStatusLists.#methodGHL[#tempIndex];
	              EXIT;
	            END_IF;
	          END_FOR;
	          #statOpcUaRequests.methodsGHL := FALSE;
	          // Count up statRegisterCount
	          #statDiagCounter.RegisterMethods += 1;
	          // Nodes are registered
	          #statRegisteredLists.Methods := TRUE;
	        END_IF;
	      END_REGION
	      
	    END_REGION
	    
	  #STATE_CONNECTED:
	    
	    REGION Command and Idle
	      //Idle as long as no Command was triggered
	      IF NOT #statBusy AND NOT #read AND NOT #write AND NOT #callMethod AND NOT #statCheckConnectionStatus THEN
	        #statDone := FALSE;
	        #statDiagnostics.status := #STATUS_IDLE;
	      END_IF;
	      //OPC_UA_GetStatus function is called cyclically, so the connection is monitored
	      #instCycDiag.TON(IN := NOT #statCycDiagTrigger,
	                       PT := #CYC_TIME_GCS);
	      #statCycDiagTrigger := FALSE;
	      IF #instCycDiag.Q AND NOT #statRHLTrigger AND NOT #tempDisconnectTrigger THEN
	        #statCheckConnectionStatus := TRUE;
	        #statCycDiagTrigger := TRUE;
	      END_IF;
	      
	      REGION Read
	        //Trigger if nodes are registered
	        IF #statRegisteredLists.Read AND #statConnected THEN
	          #tempReadTrigger := #read AND NOT #statOldTriggers.read;
	          #statOldTriggers.read := #read;
	        ELSE
	          IF #read AND #statConnected THEN
	            #statDiagnostics.status := #ERR_RL_NOTREG; //Error no ReadList is registerd Request denied
	            #statDiagnostics.subfunctionStatus := #STATUS_NOT_REGISTERED;
	          ELSE
	            IF NOT #statCheckConnectionStatus THEN
	              #statDiagnostics.status := #STATUS_IDLE; //Wait for Connection Get Status
	            END_IF;
	          END_IF;
	        END_IF;
	        
	        IF #tempReadTrigger THEN
	          #statOpcUaRequests.read := TRUE;
	          #statBusy := TRUE;
	          #statDiagnostics.status := #STATUS_BUSY;
	        ELSE
	          #statOpcUaRequests.read := FALSE;
	        END_IF;
	        //Error
	        IF #instOpcUaReadList.Error THEN
	          //--> Call ConnectionGetStatus if Status = "16#800D0000"
	          IF #instOpcUaReadList.Status = #STATUS_SERVER_NOT_CONNECTED THEN
	            #statCheckConnectionStatus := TRUE;
	          END_IF;
	          #statOpcUaRequests.read := FALSE;
	          // => OUT
	          #statBusy := FALSE;
	          #statDiagnostics.status := #ERR_RL;
	          #statDiagnostics.subfunctionStatus := #instOpcUaReadList.Status;
	        END_IF;
	        
	        //Done
	        IF #instOpcUaReadList.Done THEN
	          //Check StatusList
	          FOR #tempIndex := 0 TO UDINT_TO_INT(CountOfElements(#readNodeIds) - 1) DO
	            IF #statOpcUaStatusLists.#readList[#tempIndex] <> 16#0 THEN
	              // => OUT
	              #statDone := FALSE;
	              #statBusy := FALSE;
	              #statDiagnostics.status := #ERR_RL_SL;
	              #statDiagnostics.subfunctionStatus := #statOpcUaStatusLists.readList[#tempIndex];
	              EXIT;
	            END_IF;
	          END_FOR;
	          #statOpcUaRequests.read := FALSE;
	          // => OUT
	          IF NOT #statDiagnostics.status.%X15 THEN
	            #statDone := TRUE;
	            #statBusy := FALSE;
	            #statDiagnostics.status := #STATUS_DONE;
	            //Count up statReadCount
	            #statDiagCounter.Read += 1;
	            //--> Nodes are read continously ...
	          END_IF;
	        END_IF;
	      END_REGION
	      
	      REGION Write
	        //Trigger if nodes are registered
	        IF #statRegisteredLists.Write AND #statConnected THEN
	          #tempWriteTrigger := #write AND NOT #statOldTriggers.write;
	          #statOldTriggers.write := #write;
	        ELSE
	          IF #write AND #statConnected THEN
	            #statDiagnostics.status := #ERR_WL_NOTREG; //Error no WriteList is registerd Request denied
	            #statDiagnostics.subfunctionStatus := #STATUS_NOT_REGISTERED;
	          ELSE
	            IF NOT #statCheckConnectionStatus THEN
	              #statDiagnostics.status := #STATUS_IDLE; //Wait for Connection Get Status
	            END_IF;
	          END_IF;
	        END_IF;
	        
	        IF #tempWriteTrigger THEN
	          #statOpcUaRequests.write := TRUE;
	          #statBusy := TRUE;
	          #statDiagnostics.status := #STATUS_BUSY;
	        ELSE
	          #statOpcUaRequests.write := FALSE;
	        END_IF;
	        //Error
	        IF #instOpcUaWriteList.Error THEN
	          //--> Call ConnectionGetStatus if Status = "16#800D0000"
	          IF #instOpcUaWriteList.Status = #STATUS_SERVER_NOT_CONNECTED THEN
	            #statCheckConnectionStatus := TRUE;
	          END_IF;
	          #statOpcUaRequests.write := FALSE;
	          // => OUT
	          #statBusy := FALSE;
	          #statDiagnostics.status := #ERR_WL;
	          #statDiagnostics.subfunctionStatus := #instOpcUaWriteList.Status;
	        END_IF;
	        
	        //Done
	        IF #instOpcUaWriteList.Done THEN
	          //Check StatusList
	          FOR #tempIndex := 0 TO UDINT_TO_INT(CountOfElements(#writeNodeIds) - 1) DO
	            IF #statOpcUaStatusLists.#writeList[#tempIndex] <> 16#0 THEN
	              // => OUT
	              #statDone := FALSE;
	              #statBusy := FALSE;
	              #statDiagnostics.status := #ERR_WL_SL;
	              #statDiagnostics.subfunctionStatus := #statOpcUaStatusLists.#writeList[#tempIndex];
	              EXIT;
	            END_IF;
	          END_FOR;
	          
	          #statOpcUaRequests.write := FALSE;
	          // => OUT
	          IF NOT #statDiagnostics.status.%X15 THEN
	            #statDone := TRUE;
	            #statBusy := FALSE;
	            #statDiagnostics.status := #STATUS_DONE;
	            //Count up statwriteCount
	            #statDiagCounter.Write += 1;
	            //--> Nodes are write continously ...
	          END_IF;
	        END_IF;
	      END_REGION
	      
	      REGION Method Call
	        //Trigger if methods are registered
	        IF #statRegisteredLists.Methods AND #statConnected THEN
	          #tempMethodCallTrigger := #callMethod AND NOT #statOldTriggers.callMethod;
	          #statOldTriggers.callMethod := #callMethod;
	        ELSE
	          IF #callMethod AND #statConnected THEN
	            #statDiagnostics.status := #ERR_MC_NOTREG; //Error no MethodList is registerd Request denied
	            #statDiagnostics.subfunctionStatus := #STATUS_NOT_REGISTERED;
	          ELSE
	            IF NOT #statCheckConnectionStatus THEN
	              #statDiagnostics.status := #STATUS_IDLE; //Wait for Connection Get Status
	            END_IF;
	          END_IF;
	        END_IF;
	        
	        IF #tempMethodCallTrigger THEN
	          #statMethodHdlId := #methodHdlIndex * 0;
	          //Define statMethodHdl for the input methodHdlIndex choosen index of MethodList
	          #tempRetVal := Serialize(SRC_VARIABLE := #methodHdls,
	                                   DEST_ARRAY => #statSerializeMethodHdls,
	                                   POS := #statMethodHdlId);
	          IF #tempRetVal <> 0 THEN
	            #statDiagnostics.status := #ERR_MC_SERIALIZE;
	            #statDiagnostics.subfunctionStatus := INT_TO_WORD(#tempRetVal);
	          ELSE
	            #statMethodHdlId := #methodHdlIndex * 4;
	            #statMethodHdl.%B0 := #statSerializeMethodHdls[#statMethodHdlId + 3];
	            #statMethodHdl.%B1 := #statSerializeMethodHdls[#statMethodHdlId + 2];
	            #statMethodHdl.%B2 := #statSerializeMethodHdls[#statMethodHdlId + 1];
	            #statMethodHdl.%B3 := #statSerializeMethodHdls[#statMethodHdlId];
	            //Start Method Call
	            #statOpcUaRequests.methodCall := TRUE;
	            #statBusy := TRUE;
	            #statDiagnostics.status := #STATUS_BUSY;
	          END_IF;
	        ELSE
	          #statOpcUaRequests.methodCall := FALSE;
	        END_IF;
	        //Error
	        IF #instOpcUaMethodCall.Error THEN
	          //--> Call ConnectionGetStatus if Status = "16#800D0000"
	          IF #instOpcUaMethodCall.Status = #STATUS_SERVER_NOT_CONNECTED THEN
	            #statCheckConnectionStatus := TRUE;
	          END_IF;
	          #statOpcUaRequests.methodCall := FALSE;
	          // => OUT
	          #statBusy := FALSE;
	          #statDiagnostics.status := #ERR_MC;
	          #statDiagnostics.subfunctionStatus := #instOpcUaMethodCall.Status;
	        END_IF;
	        
	        //Done
	        IF #instOpcUaMethodCall.Done THEN
	          //Check MethodResult
	          IF #statMethodResult <> 0 THEN
	            #statBusy := FALSE;
	            #statDiagnostics.status := #ERR_MC_RESULT;
	            #statDiagnostics.subfunctionStatus := #statMethodResult;
	          END_IF;
	          #statOpcUaRequests.methodCall := FALSE;
	          // => OUT
	          #statDone := TRUE;
	          #statBusy := FALSE;
	          #statDiagnostics.status := #STATUS_DONE;
	          //Count up statwriteCount
	          #statDiagCounter.MethodCall += 1;
	          //--> Methods can be called continously ...
	        END_IF;
	      END_REGION
	      
	      REGION Disconnect Trigger
	        // Trigger to release handles if OPC UA connection should be disconnected
	        #tempClearSessionTrigger := NOT #enable AND #statOldTriggers.clearSession;
	        #statOldTriggers.clearSession := #enable;
	        
	        IF #tempClearSessionTrigger THEN
	          #statBusy := TRUE;
	          #statRHLTrigger := TRUE;
	          #statState := #STATE_DISCONNECT;
	          #statDiagnostics.status := #STATUS_BUSY;
	        END_IF;
	      END_REGION
	    END_REGION
	    
	  #STATE_DISCONNECT:
	    REGION Clear Session
	      //If Disconnect requested, release nodes -> disconnect established connection
	      //-------DISCONNECT HANDLING------------
	      //--------------------------------------
	      
	      IF #statRHLTrigger THEN
	        IF #statRegisteredLists.Write AND #writeNodeIds <> NULL AND #writeNodeHdls <> NULL THEN
	          #statOpcUaRequests.writeRHL := TRUE;
	        ELSE
	          IF #statRegisteredLists.Read AND #readNodeIds <> NULL AND #readNodeHdls <> NULL THEN
	            #statOpcUaRequests.readRHL := TRUE;
	          ELSE
	            IF #statRegisteredLists.Methods AND #methodNodeIds <> NULL AND #methodHdls <> NULL AND #objNodeIds <> NULL THEN
	              #statOpcUaRequests.methodsRHL := TRUE;
	            ELSE
	              #statRHLTrigger := FALSE;
	            END_IF;
	          END_IF;
	        END_IF;
	      END_IF;
	      REGION Release ReadList
	        //Release Handle List of Read Nodes was not successful
	        IF #InstOpcUaRHLRead.Error THEN
	          //--> Call ConnectionGetStatus if Status = "16#800D0000" or "16#80AE0000"
	          IF #InstOpcUaRHLRead.Status = #STATUS_SERVER_NOT_CONNECTED
	            OR #InstOpcUaRHLRead.Status = #STATUS_BAD_CONNECTION_CLOSED
	          THEN
	            #statCheckConnectionStatus := TRUE;
	          END_IF;
	          #statOpcUaRequests.readRHL := FALSE;
	          // => OUT
	          #statDiagnostics.status := #ERR_R_RHL;
	          #statDiagnostics.subfunctionStatus := #InstOpcUaRHLRead.Status;
	        END_IF;
	        
	        //Release Handle List of Read Nodes was successful
	        IF #InstOpcUaRHLRead.Done THEN
	          //Check StatusList
	          FOR #tempIndex := 0 TO UDINT_TO_INT(CountOfElements(#readNodeIds) - 1) DO
	            IF #statOpcUaStatusLists.#readRHL[#tempIndex] <> 16#0 THEN
	              // => OUT
	              #statDone := FALSE;
	              #statBusy := FALSE;
	              #statDiagnostics.status := #ERR_R_RHL_SL;
	              #statDiagnostics.subfunctionStatus := #statOpcUaStatusLists.readRHL[#tempIndex];
	              EXIT;
	            END_IF;
	          END_FOR;
	          #statOpcUaRequests.readRHL := FALSE;
	          #statRegisteredLists.Read := FALSE;
	          IF NOT #statDiagnostics.status.%X15 THEN
	            // => OUT
	            #statBusy := FALSE;
	            #statDiagnostics.status := #STATUS_DONE;
	            //--> Nodes are released
	          END_IF;
	        END_IF;
	      END_REGION
	      
	      REGION Release WriteList
	        //Release Handle List of Write Nodes was not successful
	        IF #instOpcUaRHLWrite.Error THEN
	          //--> Call ConnectionGetStatus if Status = "16#800D0000" or "16#80AE0000"
	          IF #instOpcUaRHLWrite.Status = #STATUS_SERVER_NOT_CONNECTED
	            OR #instOpcUaRHLWrite.Status = #STATUS_BAD_CONNECTION_CLOSED
	          THEN
	            #statCheckConnectionStatus := TRUE;
	          END_IF;
	          #statOpcUaRequests.writeRHL := FALSE;
	          // => OUT
	          #statDiagnostics.status := #ERR_W_RHL;
	          #statDiagnostics.subfunctionStatus := #instOpcUaRHLWrite.Status;
	        END_IF;
	        
	        //Release Handle List of Write Nodes was successful
	        IF #instOpcUaRHLWrite.Done THEN
	          //Check StatusList
	          FOR #tempIndex := 0 TO UDINT_TO_INT(CountOfElements(#writeNodeIds) - 1) DO
	            IF #statOpcUaStatusLists.writeRHL[#tempIndex] <> 16#0 THEN
	              // => OUT
	              #statDone := FALSE;
	              #statBusy := FALSE;
	              #statDiagnostics.status := #ERR_W_RHL_SL;
	              #statDiagnostics.subfunctionStatus := #statOpcUaStatusLists.#writeRHL[#tempIndex];
	              EXIT;
	            END_IF;
	          END_FOR;
	          #statOpcUaRequests.writeRHL := FALSE;
	          #statRegisteredLists.Write := FALSE;
	          IF NOT #statDiagnostics.status.%X15 THEN
	            // => OUT
	            #statBusy := FALSE;
	            #statDiagnostics.status := #STATUS_DONE;
	            //--> Nodes are released
	          END_IF;
	        END_IF;
	      END_REGION
	      
	      REGION Release MethodList
	        //Release Handle List of Methods was not successful
	        IF #instOpcUaRHLMethods.Error THEN
	          //--> Call ConnectionGetStatus if Status = "16#800D0000" or "16#80AE0000"
	          IF #instOpcUaRHLMethods.Status = #STATUS_SERVER_NOT_CONNECTED
	            OR #InstOpcUaRHLRead.Status = #STATUS_BAD_CONNECTION_CLOSED
	          THEN
	            #statCheckConnectionStatus := TRUE;
	          END_IF;
	          #statOpcUaRequests.methodsRHL := FALSE;
	          // => OUT
	          #statDiagnostics.status := #ERR_M_RHL;
	          #statDiagnostics.subfunctionStatus := #instOpcUaRHLMethods.Status;
	        END_IF;
	        
	        //Release Handle List of Methods was successful
	        IF #instOpcUaRHLMethods.Done THEN
	          //Check StatusList
	          FOR #tempIndex := 0 TO UDINT_TO_INT(CountOfElements(#methodNodeIds) - 1) DO
	            IF #statOpcUaStatusLists.#methodRHL[#tempIndex] <> 16#0 THEN
	              // => OUT
	              #statDone := FALSE;
	              #statBusy := FALSE;
	              #statDiagnostics.status := #ERR_M_RHL_SL;
	              #statDiagnostics.subfunctionStatus := #statOpcUaStatusLists.#methodRHL[#tempIndex];
	              EXIT;
	            END_IF;
	          END_FOR;
	          #statOpcUaRequests.methodsRHL := FALSE;
	          #statRegisteredLists.Methods := FALSE;
	          IF NOT #statDiagnostics.status.%X15 THEN
	            // => OUT
	            #statBusy := FALSE;
	            #statDiagnostics.status := #STATUS_DONE;
	            //--> Nodes are released
	          END_IF;
	        END_IF;
	      END_REGION
	      
	      REGION Disconnect
	        // disconnect trigger, if all nodes and methods are deregistered
	        #tempDisconnectTrigger := NOT #statRegisteredLists.Read AND NOT #statRegisteredLists.Write AND NOT #statRegisteredLists.Methods AND NOT #statOldTriggers.disconnect;
	        #statOldTriggers.disconnect := NOT #statRegisteredLists.Read AND NOT #statRegisteredLists.Write AND NOT #statRegisteredLists.Methods;
	        IF #tempDisconnectTrigger THEN
	          IF #statConnectionHdl <> 16#0 THEN
	            #statOpcUaRequests.disconnect := TRUE;
	            //set FB Outputs
	            #statConnectionHdl := 0;
	            #statBusy := TRUE;
	            #statDiagnostics.status := #STATUS_BUSY;
	          ELSE
	            #statState := #STATE_CONNECT;
	            //Error No connection established
	          END_IF;
	        ELSE
	          #statOpcUaRequests.disconnect := FALSE;
	        END_IF;
	        
	        //Error at connection establishment
	        IF #instOpcUaDisconnect.Error THEN
	          #statBusy := FALSE;
	          #statDiagnostics.status := #ERR_DISCON;
	          #statDiagnostics.subfunctionStatus := #instOpcUaDisconnect.Status;
	          #statCheckConnectionStatus := TRUE;
	        END_IF;
	        
	        //Disconnect was successful
	        IF #instOpcUaDisconnect.Done THEN
	          #statConnected := FALSE;
	          #statDone := FALSE;
	          #statRegisteredLists.NamespaceIndexes := FALSE;
	          #statBusy := FALSE;
	          #statOpcUaRequests.disconnect := FALSE;
	          
	          IF NOT #statDiagnostics.status.%X15 THEN
	            #statDiagnostics.status := #STATUS_DONE;
	          END_IF;
	          //reset positive edges of functions
	          #statOldTriggers.read := FALSE;
	          #statOldTriggers.write := FALSE;
	          #statOldTriggers.callMethod := FALSE;
	          #statOldTriggers.disconnect := FALSE;
	          #statOldTriggers.clearSession := FALSE;
	          #statState := #STATE_CONNECT;
	        END_IF;
	      END_REGION
	    END_REGION
	    
	  ELSE  // Statement section ELSE
	    ; //Not reachable
	END_CASE;
	REGION Connection Diagnostics
	  IF #statCheckConnectionStatus AND #enable AND (#statConnected OR #statDiagnostics.subfunctionStatus <> #CGS_CONNECTED)
	  THEN
	    #statOpcUaRequests.conGS := TRUE;
	    IF #instOpcUaConnectionGetStatus.Error THEN
	      #statOpcUaRequests.conGS := FALSE;
	      // => OUT
	      #statBusy := FALSE;
	      #statDiagnostics.status := #ERR_CGS;
	      #statDiagnostics.subfunctionStatus := #instOpcUaConnectionGetStatus.Status;
	    END_IF;
	    //Done
	    IF #instOpcUaConnectionGetStatus.Done THEN
	      //ConnectionStatus+ServerState+ServiceLevel are "Good"
	      IF #instOpcUaConnectionGetStatus.ConnectionStatus = #CGS_CONNECTED
	        AND #instOpcUaConnectionGetStatus.ServerState = #CGS_SS_RUNNING
	        AND #instOpcUaConnectionGetStatus.ServiceLevel = #CGS_SL_GOOD
	      THEN
	        REGION Connection OK
	          #statOpcUaRequests.conGS := FALSE;
	          //Session is reactivated and nodes are still registered --> Next Step --> CommandAndIdle
	          IF #statConnected AND #statRegisteredLists.NamespaceIndexes
	            AND (#statRegisteredLists.Read OR #readNodeIds = NULL)
	            AND (#statRegisteredLists.Write OR #writeNodeIds = NULL)
	            AND (#statRegisteredLists.Methods OR #methodNodeIds = NULL)
	          THEN
	            #statBusy := FALSE;
	            #statCheckConnectionStatus := FALSE;
	            //Session is reactivated and nodes are not registered yet --> Next Step --> NodeGetHandleList
	          ELSIF #statConnected AND #statRegisteredLists.NamespaceIndexes
	            AND (NOT #statRegisteredLists.Read OR NOT #statRegisteredLists.Write OR NOT #statRegisteredLists.Methods)
	          THEN
	            #statState := #STATE_NODE_GET_HANDLE_LIST;
	            #statCheckConnectionStatus := FALSE;
	            //Session is reactivated and namespaceIndexes are not set yet --> Next Step --> NamespaceGetIndexList
	          ELSIF #statConnected AND NOT #statRegisteredLists.NamespaceIndexes
	            AND (NOT #statRegisteredLists.Read OR NOT #statRegisteredLists.Write OR NOT #statRegisteredLists.Methods)
	          THEN
	            #statState := #STATE_NAMESPACE_GET_INDEX_LIST;
	            #statCheckConnectionStatus := FALSE;
	            //Session is reactivated (but connected bit isn't set) and namespaceIndexes are set and nodes are registered
	            //--> Next Step --> CommandAndIdle
	          ELSIF NOT #statConnected AND #statRegisteredLists.NamespaceIndexes
	            AND (#statRegisteredLists.Read OR #readNodeIds = NULL)
	            AND (#statRegisteredLists.Write OR #writeNodeIds = NULL)
	            AND (#statRegisteredLists.Methods OR #methodNodeIds = NULL)
	          THEN
	            //connected has to be set
	            #statConnected := TRUE;
	            #statBusy := FALSE;
	            #statRHLTrigger := FALSE;
	            #statOpcUaRequests.writeRHL := FALSE;
	            #statOpcUaRequests.readRHL := FALSE;
	            #statOpcUaRequests.methodsRHL := FALSE;
	            #statCheckConnectionStatus := FALSE;
	          END_IF;
	        END_REGION
	      ELSE
	        REGION Connection Defect
	          IF #enable THEN
	            //ConnectionStatus is in Status Connection Error -> Connection has to be monitored
	            IF #instOpcUaConnectionGetStatus.ConnectionStatus = #CGS_CONN_ERROR THEN
	              #statOpcUaRequests.conGS := FALSE;
	              // => OUT
	              #statBusy := FALSE;
	              #statConnected := FALSE;
	              #statDiagnostics.status := #ERR_CGS_CSTATE;
	              #statDiagnostics.subfunctionStatus := UDINT_TO_DWORD(#instOpcUaConnectionGetStatus.ConnectionStatus);
	              //Connection status is in Shutdown -> connection handle has to be released with OPC_UA_Disconnect
	            ELSIF #instOpcUaConnectionGetStatus.ConnectionStatus = #CGS_SHUTDOWN THEN
	              #statOpcUaRequests.conGS := FALSE;
	              #statState := #STATE_CONNECT;
	              #statRegisteredLists.Read := FALSE;
	              #statRegisteredLists.Write := FALSE;
	              #statRegisteredLists.Methods := FALSE;
	              #statCheckConnectionStatus := FALSE;
	              // => OUT
	              #statBusy := FALSE;
	              #statConnected := FALSE;
	              #statDiagnostics.status := #ERR_CGS_CSTATE_SHUTDOWN;
	              #statDiagnostics.subfunctionStatus := UDINT_TO_DWORD(#instOpcUaConnectionGetStatus.ConnectionStatus);
	              
	              //ServerState is not "Good"
	            ELSIF #instOpcUaConnectionGetStatus.ServerState <> #CGS_SS_RUNNING THEN
	              #statOpcUaRequests.conGS := FALSE;
	              // => OUT
	              #statBusy := FALSE;
	              #statConnected := FALSE;
	              #statDiagnostics.status := #ERR_CGS_SSTATE;
	              #statDiagnostics.subfunctionStatus := UDINT_TO_DWORD(#instOpcUaConnectionGetStatus.ServerState);
	              //ServiceLevel is not "Good"
	            ELSIF #instOpcUaConnectionGetStatus.ServiceLevel <> #CGS_SL_GOOD THEN
	              #statOpcUaRequests.conGS := FALSE;
	              // => OUT
	              #statBusy := FALSE;
	              #statDiagnostics.status := #ERR_CGS_SLVL;
	              #statDiagnostics.subfunctionStatus := #instOpcUaConnectionGetStatus.ServiceLevel;
	            END_IF;
	          ELSE
	            //enable is not set -> connection was faulty -> back to case CONNECT
	            //new connection can be set up
	            #statCheckConnectionStatus := FALSE;
	            #statOpcUaRequests.conGS := FALSE;
	            #statRHLTrigger := FALSE;
	            #statRegisteredLists.NamespaceIndexes := FALSE;
	            #statRegisteredLists.Read := FALSE;
	            #statRegisteredLists.Write := FALSE;
	            #statRegisteredLists.Methods := FALSE;
	          END_IF;
	        END_REGION
	      END_IF;
	    END_IF;
	  END_IF;
	END_REGION
	
	REGION Call SFBs
	  //CALL SFB OPC_UA_Connect
	  #instOpcUaConnect(REQ := #statOpcUaRequests.connect,
	                    ServerEndpointUrl := #serverEndpointUrl,
	                    SessionConnectInfo := #connectionInfo,
	                    Timeout := #OPC_UA_FUNCTIONS_TIMEOUT,
	                    ConnectionHdl => #statConnectionHdl);
	  
	  //CALL SFB OPC_UA_NamespaceGetIndexList 
	  #instOpcUaNamespaceGIL(REQ := #statOpcUaRequests.NGIL,
	                         ConnectionHdl := #statConnectionHdl,
	                         NamespaceUrisCount := UDINT_TO_UINT(CountOfElements(#namespaceUris)),
	                         NamespaceUris := #namespaceUris,
	                         Timeout := #OPC_UA_FUNCTIONS_TIMEOUT,
	                         StatusList := #statOpcUaStatusLists.#namespaceGIL,
	                         NamespaceIndexes := #namespaceIndexes);
	  
	  //CALL SFB OPC_UA_NodeGetHandleList_Read
	  #InstOpcUaGHLRead(REQ := #statOpcUaRequests.readGHL,
	                    ConnectionHdl := #statConnectionHdl,
	                    NodeIDCount := UDINT_TO_UINT(CountOfElements(#readNodeIds)),
	                    NodeIDs := #readNodeIds,
	                    Timeout := #OPC_UA_FUNCTIONS_TIMEOUT,
	                    NamespaceIndexCount := UDINT_TO_UINT(CountOfElements(#namespaceIndexes)),
	                    NamespaceIndexes := #namespaceIndexes,
	                    NodeStatusList := #statOpcUaStatusLists.#readGHL,
	                    NodeHdls := #readNodeHdls);
	  
	  //CALL SFB OPC_UA_NodeGetHandleList_Write
	  #instOpcUaGHLWrite(REQ := #statOpcUaRequests.writeGHL,
	                     ConnectionHdl := #statConnectionHdl,
	                     NodeIDCount := UDINT_TO_UINT(CountOfElements(#writeNodeIds)),
	                     NodeIDs := #writeNodeIds,
	                     Timeout := #OPC_UA_FUNCTIONS_TIMEOUT,
	                     NamespaceIndexCount := UDINT_TO_UINT(CountOfElements(#namespaceIndexes)),
	                     NamespaceIndexes := #namespaceIndexes,
	                     NodeStatusList := #statOpcUaStatusLists.#writeGHL,
	                     NodeHdls := #writeNodeHdls);
	  
	  //CALL SFB OPC_UA_MethodGetHandleList
	  #instOpcUaGHLMethods(REQ := #statOpcUaRequests.methodsGHL,
	                       ConnectionHdl := #statConnectionHdl,
	                       NodeIDCount := UDINT_TO_UINT(CountOfElements(#methodNodeIds)),
	                       ObjectNodeIDs := #objNodeIds,
	                       MethodNodeIDs := #methodNodeIds,
	                       Timeout := #OPC_UA_FUNCTIONS_TIMEOUT,
	                       NamespaceIndexCount := UDINT_TO_UINT(CountOfElements(#namespaceIndexes)),
	                       NamespaceIndexes := #namespaceIndexes,
	                       StatusList := #statOpcUaStatusLists.#methodGHL,
	                       MethodHdls := #methodHdls);
	  
	  //CALL SFB OPC_UA_ReadList
	  #instOpcUaReadList(REQ := #statOpcUaRequests.read,
	                     ConnectionHdl := #statConnectionHdl,
	                     NodeHdlCount := UDINT_TO_UINT(CountOfElements(#readNodeHdls)),
	                     NodeHdls := #readNodeHdls,
	                     Timeout := #OPC_UA_FUNCTIONS_TIMEOUT,
	                     NodeStatusList := #statOpcUaStatusLists.#readList,
	                     TimeStamps := #statOpcUaReadTimeStamps,
	                     Variable := #readData);
	  
	  //CALL SFB OPC_UA_WriteList
	  #instOpcUaWriteList(REQ := #statOpcUaRequests.write,
	                      ConnectionHdl := #statConnectionHdl,
	                      NodeHdlCount := UDINT_TO_UINT(CountOfElements(#writeNodeHdls)),
	                      NodeHdls := #writeNodeHdls,
	                      Timeout := #OPC_UA_FUNCTIONS_TIMEOUT,
	                      NodeStatusList := #statOpcUaStatusLists.#writeList,
	                      Variable := #writeData);
	  
	  //CALL SFB OPC_UA_MethodCall
	  #instOpcUaMethodCall(REQ := #statOpcUaRequests.methodCall,
	                       ConnectionHdl := #statConnectionHdl,
	                       MethodHdl := #statMethodHdl,
	                       Timeout := #OPC_UA_FUNCTIONS_TIMEOUT,
	                       MethodResult := #statMethodResult,
	                       InputArguments := #inputArguments,
	                       OutputArguments := #outputArguments);
	  
	  //CALL SFB OPC_UA_NodeReleaseHandleList_Read
	  #InstOpcUaRHLRead(REQ := #statOpcUaRequests.readRHL,
	                    ConnectionHdl := #statConnectionHdl,
	                    NodeHdlCount := UDINT_TO_UINT(CountOfElements(#readNodeHdls)),
	                    NodeHdls := #readNodeHdls,
	                    Timeout := #OPC_UA_FUNCTIONS_TIMEOUT,
	                    NodeStatusList := #statOpcUaStatusLists.#readRHL);
	  
	  //CALL SFB OPC_UA_NodeReleaseHandleList_Write
	  #instOpcUaRHLWrite(REQ := #statOpcUaRequests.writeRHL,
	                     ConnectionHdl := #statConnectionHdl,
	                     NodeHdlCount := UDINT_TO_UINT(CountOfElements(#writeNodeHdls)),
	                     NodeHdls := #writeNodeHdls,
	                     Timeout := #OPC_UA_FUNCTIONS_TIMEOUT,
	                     NodeStatusList := #statOpcUaStatusLists.#writeRHL);
	  
	  //CALL SFB OPC_UA_MethodReleaseHandleList
	  #instOpcUaRHLMethods(REQ := #statOpcUaRequests.methodsRHL,
	                       ConnectionHdl := #statConnectionHdl,
	                       MethodHdlCount := UDINT_TO_UINT(CountOfElements(#methodHdls)),
	                       MethodHdls := #methodHdls,
	                       Timeout := #OPC_UA_FUNCTIONS_TIMEOUT,
	                       StatusList := #statOpcUaStatusLists.#methodRHL);
	  
	  //CALL SFB OPC_UA_Disconnect
	  #instOpcUaDisconnect(REQ := #statOpcUaRequests.disconnect,
	                       ConnectionHdl := #statConnectionHdl,
	                       Timeout := #OPC_UA_FUNCTIONS_TIMEOUT);
	  
	  //CALL SFB OPC_UA_ConnectionGetStatus
	  #instOpcUaConnectionGetStatus(REQ := #statOpcUaRequests.conGS,
	                                ConnectionHdl := #statConnectionHdl,
	                                Timeout := #OPC_UA_FUNCTIONS_TIMEOUT);
	END_REGION
	
	REGION Set FB Outputs
	  #connected := #statConnected;
	  #done := #statDone;
	  #busy := #statBusy;
	  #error := #statDiagnostics.status.%X15;
	  #connectionHdl := #statConnectionHdl;
	  #status := #statDiagnostics.status;
	  IF #statDiagnostics.status.%X15 THEN
	    #diagnostics := #statDiagnostics;
	  END_IF;
	END_REGION
END_FUNCTION_BLOCK

FUNCTION "Extract_data_DMC" : Void   // FC2011, LAD
{ S7_Optimized_Access := 'TRUE' }
VERSION : 0.1
// stored: AutoNumber false, IsIECCheckEnabled false, SetENOAutomatically false, UDAEnableTagReadback false
   VAR_INPUT
      round : Byte;
      Data_DMC : Array[1.."MaxRoundNumber", 1..10] of "DATA_DMC";
   END_VAR
   VAR_OUTPUT
      DATA_DMC_Extract : Array[1..10] of String[25];
   END_VAR
   VAR_TEMP
      idx : SInt;
      round_idx : SInt;
   END_VAR
BEGIN

REGION Network 1
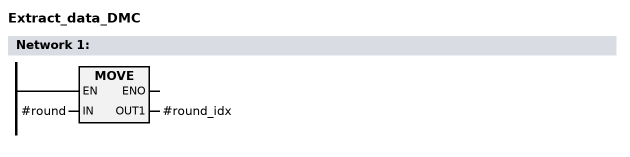
   RUNG wire#powerrail
      Move(in := #round, out1 => #round_idx)
   END_RUNG
   // the same network as SCL:
   #round_idx := #round;
END_REGION

REGION Network 2 (SCL)
   FOR  #idx:=1 TO 10 DO
       #DATA_DMC_Extract[#idx]:= #Data_DMC[#round_idx,#idx].SAP_REF_PRODUCTION;

   END_FOR;
END_REGION
END_FUNCTION

FUNCTION "Concatenate_STRING" : Void   // FC2010, LAD
{ S7_Optimized_Access := 'TRUE' }
VERSION : 0.1
// stored: AutoNumber false, IsIECCheckEnabled false, SetENOAutomatically false, UDAEnableTagReadback false
   VAR_INPUT
      DMC_SAP_REF : Array[1..10] of String[25];
   END_VAR
   VAR_OUTPUT
      String_empty : Bool;
   END_VAR
   VAR_IN_OUT
      DMC_SAP_REf_WSTRING : WString;
   END_VAR
   VAR_TEMP
      concatenate : String;
      Convert : WString;
   END_VAR
   VAR CONSTANT
      Template_string_empty : String := ';;;;;;;;;';
   END_VAR
BEGIN

REGION Network 1 (SCL): Concatenate function
       #concatenate := CONCAT(IN1 := #DMC_SAP_REF[1], IN2 := ';');
       #concatenate := CONCAT(IN1 := #concatenate, IN2 := #DMC_SAP_REF[2]);
       #concatenate := CONCAT(IN1 := #concatenate, IN2 := ';');
       #concatenate := CONCAT(IN1 := #concatenate, IN2 := #DMC_SAP_REF[3]);
       #concatenate := CONCAT(IN1 := #concatenate, IN2 := ';');
       #concatenate := CONCAT(IN1 := #concatenate, IN2 := #DMC_SAP_REF[4]);
       #concatenate := CONCAT(IN1 := #concatenate, IN2 := ';');
       #concatenate := CONCAT(IN1 := #concatenate, IN2 := #DMC_SAP_REF[5]);
       #concatenate := CONCAT(IN1 := #concatenate, IN2 := ';');
       #concatenate := CONCAT(IN1 := #concatenate, IN2 := #DMC_SAP_REF[6]);
       #concatenate := CONCAT(IN1 := #concatenate, IN2 := ';');
       #concatenate := CONCAT(IN1 := #concatenate, IN2 := #DMC_SAP_REF[7]);
       #concatenate := CONCAT(IN1 := #concatenate, IN2 := ';');
       #concatenate := CONCAT(IN1 := #concatenate, IN2 := #DMC_SAP_REF[8]);
       #concatenate := CONCAT(IN1 := #concatenate, IN2 := ';');
       #concatenate := CONCAT(IN1 := #concatenate, IN2 := #DMC_SAP_REF[9]);
       #concatenate := CONCAT(IN1 := #concatenate, IN2 := ';');
       #concatenate := CONCAT(IN1 := #concatenate, IN2 := #DMC_SAP_REF[10]);
END_REGION

REGION Network 2
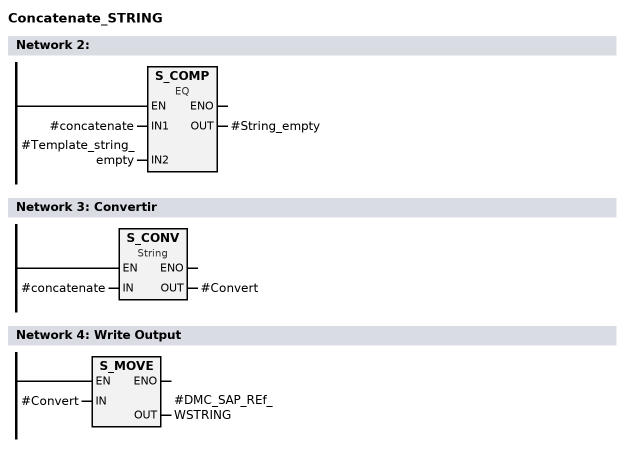
   RUNG wire#powerrail
      { S7_Templates := "[relation := EQ, src_type := String]" } S_COMP(IN1 := #concatenate, IN2 := #Template_string_empty, OUT => #String_empty)
   END_RUNG
   // the same network as SCL:
   S_COMP(IN1 := #concatenate, IN2 := #Template_string_empty, OUT => #String_empty);
END_REGION

REGION Network 3: Convertir
   RUNG wire#powerrail
      { S7_Templates := "[src_type := String, dest_type := WString]" } S_CONV(IN := #concatenate, OUT => #Convert)
   END_RUNG
   // the same network as SCL:
   S_CONV(IN := #concatenate, OUT => #Convert);
END_REGION

REGION Network 4: Write Output
   RUNG wire#powerrail
      S_Move(in := #Convert, out => #DMC_SAP_REf_WSTRING)
   END_RUNG
   // the same network as SCL:
   #DMC_SAP_REf_WSTRING := #Convert;
END_REGION
END_FUNCTION

FUNCTION_BLOCK "2. Call_M000_PRODUCTION_DECLARATION"   // FB2002, LAD
{ S7_Optimized_Access := 'TRUE' }
VERSION : 0.1
// stored: AutoNumber false, IsIECCheckEnabled false, IsRetainMemResEnabled false, MemoryReserve 100, SetENOAutomatically false, UDAEnableTagReadback false
   VAR_INPUT
      CYCLE_COUNTER : DInt;
   END_VAR
   VAR_IN_OUT
      LOCAL_PART_ARRAY : Variant;
      LOCAL_PART_WSTRING : Variant;
      LOCAL_TOOL : Variant;
      TRACA_REF : Variant;
      QUANTITY : Variant;
      STATION_NAME : Variant;   // Follow the example ST1, ST2, ST3, ST4...
   END_VAR
   VAR
      cycleCounter_temp : DInt;
      LOCAL_PART_OK : WString;
      STATION_NAME_OK : WString;
      aux : Struct
         idx : UInt;
         cnt : UInt;
         sizeCnt : Bool;
         LOCAL_PART_STRING : String;
      END_STRUCT;
   END_VAR
   VAR_TEMP
      retVal : Int;
   END_VAR
BEGIN

REGION Network 1 (SCL): PREPARE LOCAL_PART
   REGION PREPARE LOCAL_PART_ARRAY
       //Local part management - variable can be either wstring OR array of char
       IF #LOCAL_PART_WSTRING <> NULL THEN
           VariantGet(SRC := #LOCAL_PART_WSTRING,
                      DST => #LOCAL_PART_OK);
       ELSE
           IF #LOCAL_PART_ARRAY <> NULL THEN
               #aux.sizeCnt := FALSE;
               //If array of char, the array pass through a filter to delete empty positions
               Chars_TO_Strg(Chars := #LOCAL_PART_ARRAY,
                             pChars := 0,
                             Cnt := 0, //Copy all positions of char array
                             Strg => #aux.LOCAL_PART_STRING);

               //Find the last valid char
               #aux.idx := INT_TO_UINT(LEN(#aux.LOCAL_PART_STRING));

               WHILE #aux.sizeCnt = FALSE DO
                   IF #aux.LOCAL_PART_STRING[#aux.idx] <> ' ' THEN
                       //Set the index of last valid char
                       #aux.cnt := #aux.idx;
                       #aux.sizeCnt := TRUE;
                   ELSE
                       #aux.idx := #aux.idx - 1;
                   END_IF;
               END_WHILE;

               //Convert the array of char in string
               Chars_TO_Strg(Chars := #LOCAL_PART_ARRAY,
                             pChars := 0,
                             Cnt := #aux.cnt, //Copy only the right amount of data
                             Strg => #aux.LOCAL_PART_STRING);
               #LOCAL_PART_OK := STRING_TO_WSTRING(#aux.LOCAL_PART_STRING);
           ELSE
               //"MII_Parameters".M000_Status.error := TRUE;
               "MII_Parameters".M000_Status.status := WSTRING#'NO LOCAL PART DEFINED';
           END_IF;
       END_IF;
   END_REGION
END_REGION

REGION Network 2 (SCL): PREPARE CALL METHOD
   IF #cycleCounter_temp <> #CYCLE_COUNTER THEN
       #cycleCounter_temp := #CYCLE_COUNTER;

       IF #CYCLE_COUNTER > 0 THEN
           //Normal mode
           IF "MII_Parameters".Connection_Status.opcUaConnected THEN

               //Start attempts counter 
               "MII_Parameters".Connection_Status.aux.nAttemptsTotal := 1;

               //Set argument parameters
               "MII_Interface_Data".MII_METHODS.M000_PRODUCTION_DECLARATION.Inputs.CYCLE_COUNTER := DINT_TO_WSTRING(#CYCLE_COUNTER);

               "MII_Interface_Data".MII_METHODS.M000_PRODUCTION_DECLARATION.Inputs.LOCAL_PART := #LOCAL_PART_OK;

               IF #STATION_NAME <> NULL  THEN
                   // When there are more than one station at the machine, the _STn is concatenated to the PLC_ID
                   VariantGet(SRC := #STATION_NAME,
                              DST => #STATION_NAME_OK);
                   IF #STATION_NAME_OK <> WSTRING#'' THEN
                       "MII_Interface_Data".MII_METHODS.M000_PRODUCTION_DECLARATION.Inputs.PLC_ID := CONCAT_WSTRING(IN1 := "MII_Parameters".Connection.PLC_ID, IN2 := WSTRING#'_', IN3 := #STATION_NAME_OK);
                   ELSE
                       "MII_Interface_Data".MII_METHODS.M000_PRODUCTION_DECLARATION.Inputs.PLC_ID := "MII_Parameters".Connection.PLC_ID;
                   END_IF;
               ELSE
                   "MII_Interface_Data".MII_METHODS.M000_PRODUCTION_DECLARATION.Inputs.PLC_ID := "MII_Parameters".Connection.PLC_ID;
               END_IF;

               // Set PLC_ID correctly accordingly to application
               IF NOT "MII_Parameters".Connection.OperationMode THEN
                   "MII_Interface_Data".MII_METHODS.M000_PRODUCTION_DECLARATION.Inputs.PLANT := "MII_Parameters".Connection.PlantID;
               ELSE
                   "MII_Interface_Data".MII_METHODS.M000_PRODUCTION_DECLARATION.Inputs.PLANT := CONCAT(IN1 := "MII_Parameters".Connection.PlantID, IN2 := WSTRING#'_TEST');
               END_IF;

               VariantGet(SRC := #LOCAL_TOOL,
                          DST => "MII_Interface_Data".MII_METHODS.M000_PRODUCTION_DECLARATION.Inputs.LOCAL_TOOL);
               VariantGet(SRC := #TRACA_REF, 
                          DST => "MII_Interface_Data".MII_METHODS.M000_PRODUCTION_DECLARATION.Inputs.TRACA_REF);
               VariantGet(SRC := #QUANTITY,
                          DST => "MII_Interface_Data".MII_METHODS.M000_PRODUCTION_DECLARATION.Inputs.QUANTITY);

               //Set index to Production Declaration
               "1. DMC_setConnection_DB".CallBuffer[0] := TRUE;
               "MII_Parameters".M000_Status.status := WSTRING#'IN PROGRESS';

               //Downgraded mode            
           ELSE
               //Set argument parameters
               "MII_Parameters".M000_Status.Inputs.CYCLE_COUNTER := DINT_TO_WSTRING(#CYCLE_COUNTER);
               "MII_Parameters".M000_Status.Inputs.PLANT := "MII_Parameters".Connection.PlantID;
               "MII_Parameters".M000_Status.Inputs.PLC_ID := "MII_Parameters".Connection.PLC_ID;
               "MII_Parameters".M000_Status.Inputs.LOCAL_PART := #LOCAL_PART_OK;

               VariantGet(SRC := #LOCAL_TOOL,
                          DST => "MII_Parameters".M000_Status.Inputs.LOCAL_TOOL);
               VariantGet(SRC := #TRACA_REF,
                          DST => "MII_Parameters".M000_Status.Inputs.TRACA_REF);
               VariantGet(SRC := #QUANTITY,
                          DST => "MII_Parameters".M000_Status.Inputs.QUANTITY);

               //HMI MUST RESET THE VARIABLE AFTER STORING THE VALUES
               "MII_Parameters".M000_Status.error := TRUE;
               "MII_Parameters".M000_Status.status := Wstring#'DOWNGRADED';
               #retVal := RD_LOC_T("MII_Parameters".M000_Status.timestamp);
           END_IF;
       END_IF;
   END_IF;
END_REGION

REGION Network 3 (SCL): TEST MODE
   // Send pre defined data to DMC to test the communication and declaration
   IF "MII_Parameters".Commands.testProdDeclaration THEN

        //Start attempts counter 
       "MII_Parameters".Connection_Status.aux.nAttemptsTotal := 1;

       //Set standard test arguments
       "MII_Interface_Data".MII_METHODS.M000_PRODUCTION_DECLARATION.Inputs.CYCLE_COUNTER := INT_TO_WSTRING("MII_Parameters".Commands.auxTestProdDeclaration);
       "MII_Interface_Data".MII_METHODS.M000_PRODUCTION_DECLARATION.Inputs.PLANT := CONCAT(IN1 := "MII_Parameters".Connection.PlantID, IN2 := WSTRING#'_TEST');
       "MII_Interface_Data".MII_METHODS.M000_PRODUCTION_DECLARATION.Inputs.PLC_ID := "MII_Parameters".Connection.PLC_ID;
       "MII_Interface_Data".MII_METHODS.M000_PRODUCTION_DECLARATION.Inputs.LOCAL_PART := #LOCAL_PART_OK;

       "1. DMC_setConnection_DB".CallBuffer[0] := TRUE;
       "MII_Parameters".M000_Status.status := WSTRING#'IN PROGRESS';
   END_IF;
END_REGION
END_FUNCTION_BLOCK

FUNCTION_BLOCK "6. Call_M004_NTRS"   // FB2006, LAD
{ S7_Optimized_Access := 'TRUE' }
VERSION : 0.1
// stored: AutoNumber false, IsIECCheckEnabled false, IsRetainMemResEnabled false, MemoryReserve 100, SetENOAutomatically false, UDAEnableTagReadback false
   VAR_INPUT
      nTRSTag : Bool;
   END_VAR
   VAR
      nTRSTagTemp : Bool;
   END_VAR
BEGIN

REGION Network 1 (SCL)
   IF #nTRSTag <> #nTRSTagTemp THEN

       "MII_Interface_Data".MII_METHODS.M004_NTRS.Inputs.PLC_ID := "MII_Parameters".Connection.PLC_ID;
       "MII_Interface_Data".MII_METHODS.M004_NTRS.Inputs.PLANT := "MII_Parameters".Connection.PlantID;
       "MII_Interface_Data".MII_METHODS.M004_NTRS.Inputs.STOPPAGE := #nTRSTag;
       "MII_Interface_Data".MII_METHODS.M004_NTRS.Inputs.CAUSE := WSTRING#'1S014040';
       //Call the method 
       "1. DMC_setConnection_DB".CallBuffer[6] := TRUE;

       #nTRSTagTemp := #nTRSTag;
   END_IF;
END_REGION
END_FUNCTION_BLOCK

FUNCTION_BLOCK "7. Call_M103_PY"   // FB2007, LAD
{ S7_Optimized_Access := 'TRUE' }
VERSION : 0.1
// stored: AutoNumber false, IsIECCheckEnabled false, IsRetainMemResEnabled false, MemoryReserve 100, SetENOAutomatically false, UDAEnableTagReadback false
   VAR_INPUT
      PY_ON { ExternalAccessible := 'False'; ExternalVisible := 'False'; ExternalWritable := 'False'} : Bool;
      PY_DOWN { ExternalAccessible := 'False'; ExternalVisible := 'False'; ExternalWritable := 'False'} : Bool;
      PY_OFF { ExternalAccessible := 'False'; ExternalVisible := 'False'; ExternalWritable := 'False'} : Bool;
   END_VAR
   VAR
      PYOnTemp : Bool;
      PYDownTemp : Bool;
      PYOffTemp : Bool;
   END_VAR
BEGIN

REGION Network 1 (SCL)
   IF (#PY_ON <> #PYOnTemp OR #PY_DOWN <> #PYDownTemp OR #PY_OFF <> #PYOffTemp) AND (#PY_ON OR #PY_DOWN OR #PY_OFF) THEN

       "MII_Interface_Data".MII_METHODS.M103_PY.Inputs.PLC_ID := "MII_Parameters".Connection.PLC_ID;
       "MII_Interface_Data".MII_METHODS.M103_PY.Inputs.PLANT := "MII_Parameters".Connection.PlantID;

       "MII_Interface_Data".MII_METHODS.M103_PY.Inputs.PY_ON := #PY_ON;
       "MII_Interface_Data".MII_METHODS.M103_PY.Inputs.PY_DOWN := #PY_DOWN;
       "MII_Interface_Data".MII_METHODS.M103_PY.Inputs.PY_OFF := #PY_OFF;

       //Call the method 
       "1. DMC_setConnection_DB".CallBuffer[7] := TRUE;

       #PYOnTemp := #PY_ON;
       #PYDownTemp := #PY_DOWN;
       #PYOffTemp := #PY_OFF;
   END_IF;
END_REGION
END_FUNCTION_BLOCK

FUNCTION "FC_Variability" : Void   // FC2013, LAD
{ S7_Optimized_Access := 'TRUE' }
VERSION : 0.1
// V1 : Creation YM 7/04/2023
// stored: AutoNumber false, IsIECCheckEnabled false, SetENOAutomatically false, UDAEnableTagReadback false
   VAR_TEMP
      i : Int;
      j : Bool;
      result : String;
      dintLeft : DInt;
   END_VAR
BEGIN

REGION Network 1 (SCL): Convert Errors
   // FOR #i := 1 TO 32 DO
   //      "DB_Variability".ERROR[#i].%W0 := "DB_MESSAGE".ERROR_TO_HMI[(#i*2)-1];
   //      "DB_Variability".ERROR[#i].%W1 := "DB_MESSAGE".ERROR_TO_HMI[#i * 2];
   //  END_FOR;

   // FOR #i := 1 TO 32 DO
   //     // Move Error to left to remove error 0 not used on Welding cell compare standard of variability
   //     #dintLeft := SHL_DINT(IN := "DB_Variability".ERROR[#i], N := 1);
   //     //Convert Dint to String
   //     #result := "LGF_IntToString"(#dintLeft);
   //     //Convert String to wtring
   //     "DB_Variability".ERROR_TO_OPC[#i] := STRING_TO_WSTRING(#result);

   // END_FOR;
END_REGION
END_FUNCTION

FUNCTION_BLOCK "5. Call_M005_VARIABILITY"
{ S7_Optimized_Access := 'TRUE' }
VERSION : 0.1
   VAR_INPUT 
      equipmentVariability : WString;
      errorDInt : Array[1..32] of DInt;
      errorWString : Array[1..32] of WString;
      x : Bool;
   END_VAR

   VAR 
      variabilityIndex { ExternalAccessible := 'False'; ExternalVisible := 'False'; ExternalWritable := 'False'} : Array[1..32] of WString[1] := [WSTRING#'0', WSTRING#'1', WSTRING#'2', WSTRING#'3', WSTRING#'4', WSTRING#'5', WSTRING#'6', WSTRING#'7', WSTRING#'8', WSTRING#'9', WSTRING#'A', WSTRING#'B', WSTRING#'C', WSTRING#'D', WSTRING#'E', WSTRING#'F', WSTRING#'G', WSTRING#'H', WSTRING#'I', WSTRING#'J', WSTRING#'K', WSTRING#'L', WSTRING#'M', WSTRING#'N', WSTRING#'O', WSTRING#'P', WSTRING#'Q', WSTRING#'R', WSTRING#'S', WSTRING#'T', WSTRING#'U', WSTRING#'V'];
      actualValue : Array[1..32] of DInt;
      timestamp {InstructionName := 'DTL'; LibVersion := '1.0'} : DTL;
      timestampStr : Struct
         year : WString;
         month : WString;
         day : WString;
         hour : WString;
         minute : WString;
         second : WString;
      END_STRUCT;
      datestring : String;
   END_VAR

   VAR_TEMP 
      i : Int;
      ret : Int;
   END_VAR


BEGIN
	#ret := RD_LOC_T(#timestamp);
	// convert Date/hour to string
	    
	#datestring:= "LGF_DTLtoString_ISO"("date":=#timestamp, separator:='-');
	#datestring := REPLACE(IN1 := #datestring, IN2 := 'T',L:=1, P := 11);
	
	
	"MII_Interface_Data".MII_METHODS.M005_VARIABILITY.Inputs.PLC_ID := "MII_Parameters".Connection.PLC_ID;
	"MII_Interface_Data".MII_METHODS.M005_VARIABILITY.Inputs.PLANT := "MII_Parameters".Connection.PlantID;
	
	FOR #i := 1 TO 32 DO
	    IF #errorDInt[#i] <> #actualValue[#i] AND NOT "1. DMC_setConnection_DB".CallBuffer[8] THEN
	        
	        IF #x THEN
	            "MII_Interface_Data".MII_METHODS.M005_VARIABILITY.Inputs.VARIABILITY_CODE := CONCAT_WSTRING(IN1 := #equipmentVariability,
	                                                                                                        IN2 := #variabilityIndex[#i],
	                                                                                                        IN3 := WSTRING#'x');
	        ELSE
	            "MII_Interface_Data".MII_METHODS.M005_VARIABILITY.Inputs.VARIABILITY_CODE := CONCAT_WSTRING(IN1 := #equipmentVariability,
	                                                                                                        IN2 := #variabilityIndex[#i],
	                                                                                                        IN3 := WSTRING#'0');
	        END_IF;
	        
	        
	        "MII_Interface_Data".MII_METHODS.M005_VARIABILITY.Inputs.STATUS := #errorWString[#i];
	        
	        //Get error timestamp 
	        "MII_Interface_Data".MII_METHODS.M005_VARIABILITY.Inputs.TIMESTAMP := MID(IN:=STRING_TO_WSTRING(#datestring), L:=19, P:=1);
	        
	        #actualValue[#i] := #errorDInt[#i];
	        //Call the method 
	        "1. DMC_setConnection_DB".CallBuffer[8] := TRUE;
	        
	        EXIT;
	        
	    END_IF;
	END_FOR;
	
END_FUNCTION_BLOCK

FUNCTION_BLOCK "ModeSelection"   // FB38, GRAPH
VERSION : 0.1
// stored: AcknowledgeErrorsRequired true, AutoNumber true, GraphVersion 6.0, InitialValuesAcquisition false, IsIECCheckEnabled false, LanguageInNetworks LAD, LockOperatingMode false, PermanentILProcessingInMANMode false, SetENOAutomatically false, SkipSteps false, UDAEnableTagReadback false, WithAlarmHandling true
   // inherited from GRAPH_BASE
   VAR
      OFF_SQ_BASE : Bool;
   END_VAR
   VAR_INPUT
      iSafetyOKauto : Bool;
      iSafetyOKmanual : Bool;
      iBasePosition : Bool;
      iPozadavekZastavitOdDveri : Bool;
      iLinkaZastavena : Bool;
      iLinkaPrazdna : Bool;
      iBaseInManualMode : Bool;
      OFF_SQ { ExternalAccessible := 'False'; ExternalVisible := 'False'; ExternalWritable := 'False'} : Bool := false;   // Turn sequence off
      INIT_SQ { ExternalAccessible := 'False'; ExternalVisible := 'False'; ExternalWritable := 'False'} : Bool := false;   // Set sequence to initial state
      ACK_EF { ExternalAccessible := 'False'; ExternalVisible := 'False'; ExternalWritable := 'False'} : Bool := false;   // Acknowledge all errors and faults
      S_PREV { ExternalAccessible := 'False'; ExternalVisible := 'False'; ExternalWritable := 'False'} : Bool := false;   // Output previous step in parameter S_NO
      S_NEXT { ExternalAccessible := 'False'; ExternalVisible := 'False'; ExternalWritable := 'False'} : Bool := false;   // Indicate next step in parameter S_NO
      SW_AUTO { ExternalAccessible := 'False'; ExternalVisible := 'False'; ExternalWritable := 'False'} : Bool := false;   // Automatic mode
      SW_TAP { ExternalAccessible := 'False'; ExternalVisible := 'False'; ExternalWritable := 'False'} : Bool := false;   // Semiautomatic/switch with transition
      SW_TOP { ExternalAccessible := 'False'; ExternalVisible := 'False'; ExternalWritable := 'False'} : Bool := false;   // Semiautomatic/ignore transition
      SW_MAN { ExternalAccessible := 'False'; ExternalVisible := 'False'; ExternalWritable := 'False'} : Bool := false;   // Manual mode
      S_SEL { ExternalAccessible := 'False'; ExternalVisible := 'False'; ExternalWritable := 'False'} : Int := 0;   // Select step to be output to S_NO
      S_ON { ExternalAccessible := 'False'; ExternalVisible := 'False'; ExternalWritable := 'False'} : Bool := false;   // Activate step indicated in S_NO
      S_OFF { ExternalAccessible := 'False'; ExternalVisible := 'False'; ExternalWritable := 'False'} : Bool := false;   // Deactivate step indicated S_NO
      T_PUSH { ExternalAccessible := 'False'; ExternalVisible := 'False'; ExternalWritable := 'False'} : Bool := false;   // Enable transition to switch in semi automatic mode
   END_VAR
   VAR_OUTPUT
      S_NO { ExternalAccessible := 'False'; ExternalVisible := 'False'; ExternalWritable := 'False'} : Int := 0;   // Step number
      S_MORE { ExternalAccessible := 'False'; ExternalVisible := 'False'; ExternalWritable := 'False'} : Bool := false;   // More steps are available and can be shown in S_NO
      S_ACTIVE { ExternalAccessible := 'False'; ExternalVisible := 'False'; ExternalWritable := 'False'} : Bool := false;   // Step indicated in S_NO is active
      ERR_FLT { ExternalAccessible := 'False'; ExternalVisible := 'False'; ExternalWritable := 'False'} : Bool := false;   // Interlock or supervision group error
      AUTO_ON { ExternalAccessible := 'False'; ExternalVisible := 'False'; ExternalWritable := 'False'} : Bool := false;   // Automatic mode is active
      TAP_ON { ExternalAccessible := 'False'; ExternalVisible := 'False'; ExternalWritable := 'False'} : Bool := false;   // Semiautomatic mode/step with transition enabled
      TOP_ON { ExternalAccessible := 'False'; ExternalVisible := 'False'; ExternalWritable := 'False'} : Bool := false;   // Semiautomatic mode/ignore transition enabled
      MAN_ON { ExternalAccessible := 'False'; ExternalVisible := 'False'; ExternalWritable := 'False'} : Bool := false;   // Manual mode is active
   END_VAR
   VAR
      dummy : Bool;
   END_VAR
   VAR RETAIN
      mode : "udtModes";
   END_VAR
   VAR
      PrevMode : Int;
      F_TRIG_semiauto_switch { S7_SetPoint := 'True'} : F_TRIG;
      F_TRIG_switchAuto { S7_SetPoint := 'True'} : F_TRIG;
   END_VAR
BEGIN
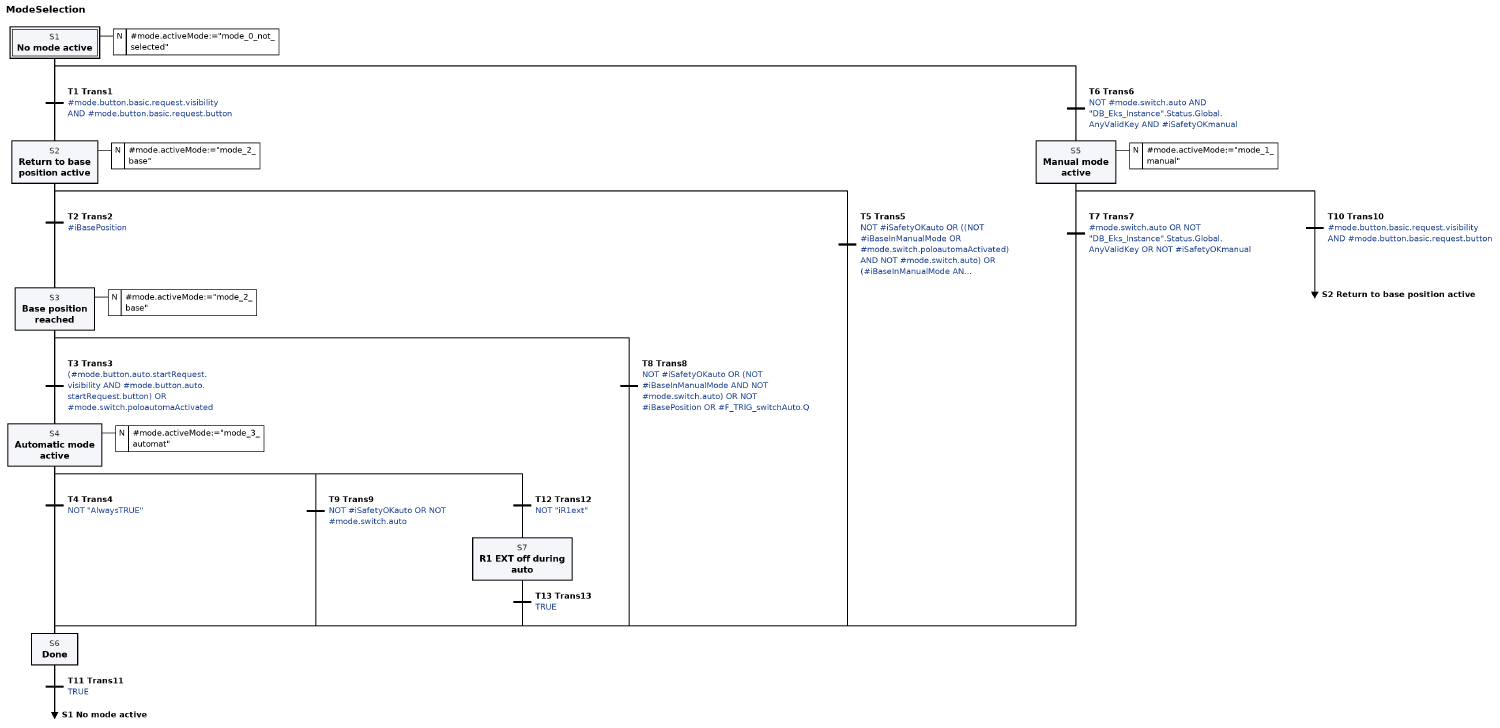
   // permanent pre-instructions
   NETWORK 1
   TITLE = mode init
      "ModeSelection_DB".mode.activeMode := "mode_0_not_selected";
   NETWORK 2
   TITLE = button visibility
      #mode.button.basic.request.visibility := #iSafetyOKauto AND ((#mode.switch.auto AND #"No mode active".X AND (NOT #iBaseInManualMode OR #mode.switch.poloautomaActivated)) OR (NOT #mode.switch.auto AND #"Manual mode active".X AND #iBaseInManualMode AND NOT #mode.switch.poloautomaActivated));
      #mode.button.auto.startRequest.visibility := #iSafetyOKauto AND #mode.switch.auto AND #"Base position reached".X AND NOT "SystemHMI".AlarmActive;
   NETWORK 3
   TITLE = semiauto switch off detection
      #F_TRIG_semiauto_switch(CLK := #mode.switch.poloautomaActivated);   // F_TRIG
   NETWORK 4
      #F_TRIG_switchAuto(CLK := #mode.switch.auto);   // F_TRIG

